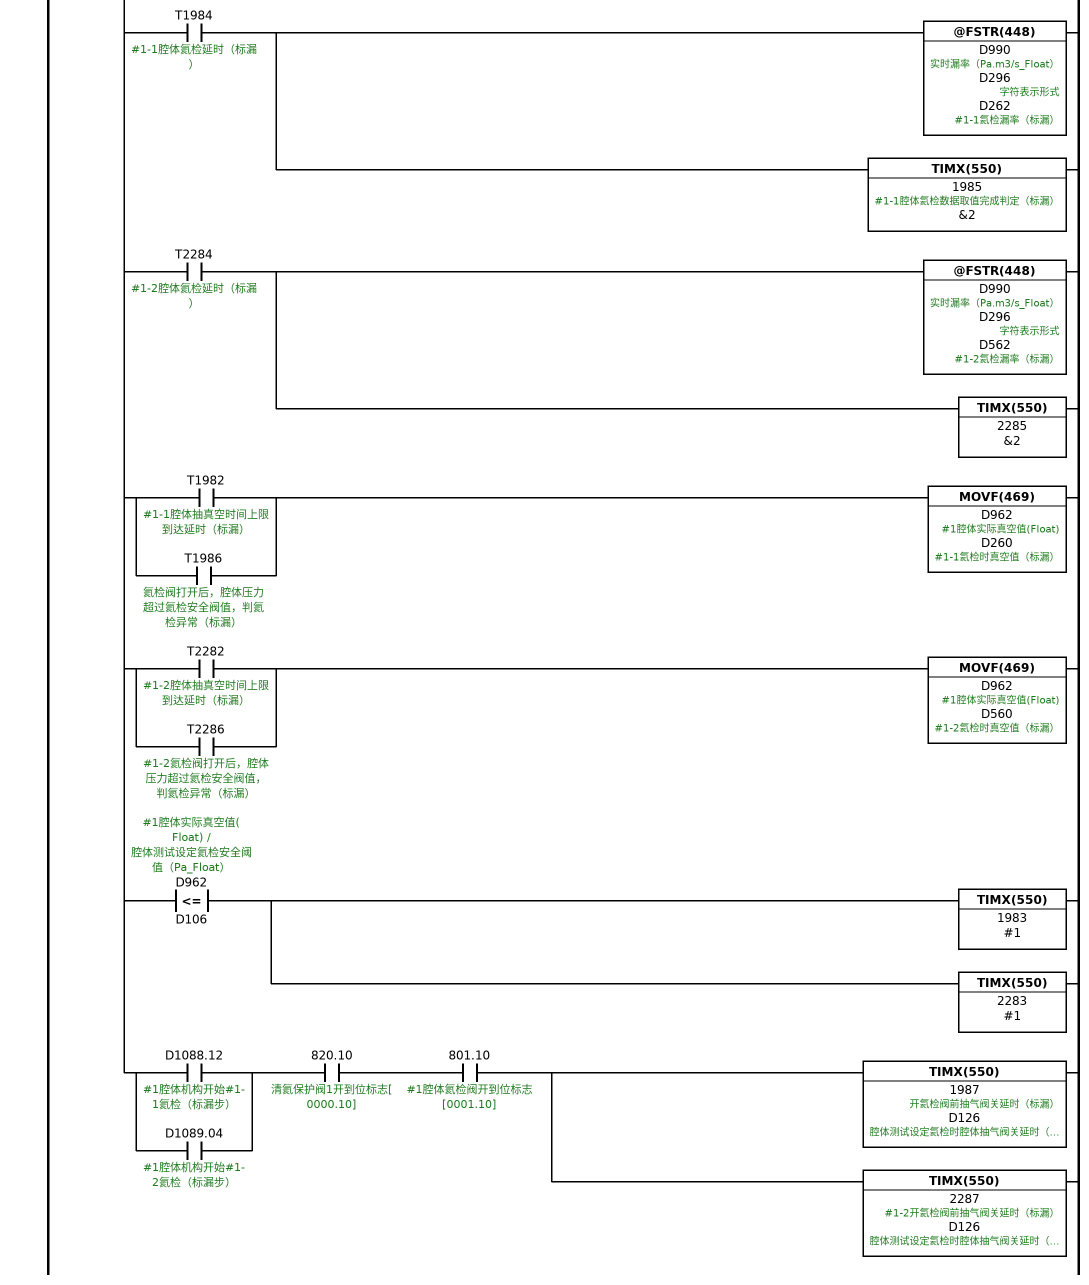
; rung 10: 标漏测试数据处理
LD P_On
OUT TR0
LD D1088.08  ; #1腔体机构开#1腔抽气阀（标漏步）
AND 821.00  ; #1腔体破真空挡板阀开到位标志
LD D1089.00  ; #1腔体机构开#1腔抽真空阀（标漏步）
AND 821.02  ; #1-2腔体阀开到位标志
ORLD
ANDLD
AND 820.14  ; #1腔体抽真空阀开到位标志
AND<=F(332) D962 D100  ; #1腔体实际真空值(Float), 腔体测试设定真空阈值（Pa_Float）
TIMX(550) 1981 &0  ; #1-1腔体抽真空阀值到达延时（标漏）
TIMX(550) 2281 &0  ; #1-2腔体抽真空阀值到达延时（标漏）
LD TR0
LD D1088.08  ; #1腔体机构开#1腔抽气阀（标漏步）
AND 821.00  ; #1腔体破真空挡板阀开到位标志
LD D1089.00  ; #1腔体机构开#1腔抽真空阀（标漏步）
AND 821.02  ; #1-2腔体阀开到位标志
ORLD
ANDLD
AND 820.14  ; #1腔体抽真空阀开到位标志
AND>F(333) D962 D100  ; #1腔体实际真空值(Float), 腔体测试设定真空阈值（Pa_Float）
TIMX(550) 1982 D102  ; 腔体测试设定抽真空时间上限（S_UInt）, #1-1腔体抽真空时间上限到达延时（标漏）
TIMX(550) 2282 D102  ; 腔体测试设定抽真空时间上限（S_UInt）, #1-2腔体抽真空时间上限到达延时（标漏）
LD TR0
AND D1088.12  ; #1腔体机构开始#1-1氦检（标漏步）
AND 821.00  ; #1腔体破真空挡板阀开到位标志
AND 820.10  ; 清氦保护阀1开到位标志[0000.10]
AND 801.10  ; #1腔体氦检阀开到位标志[0001.10]
TIMX(550) 1984 D110  ; 腔体测试设定氦检时间（S_UInt）, #1-1腔体氦检延时（标漏）
@MOVF(469) D962 D260  ; #1腔体实际真空值(Float), #1-1氦检时真空值（标漏）
AND>F(333) D962 D106  ; #1腔体实际真空值(Float), 腔体测试设定氦检安全阈值（Pa_Float）
TIMX(550) 1986 &0  ; 氦检阀打开后，腔体压力超过氦检安全阀值，判氦检异常（标漏）
LD TR0
AND D1089.04  ; #1腔体机构开始#1-2氦检（标漏步）
AND 821.02  ; #1-2腔体阀开到位标志
AND 820.10  ; 清氦保护阀1开到位标志[0000.10]
AND 801.10  ; #1腔体氦检阀开到位标志[0001.10]
TIMX(550) 2284 D110  ; 腔体测试设定氦检时间（S_UInt）, #1-2腔体氦检延时（标漏）
@MOVF(469) D962 D560  ; #1腔体实际真空值(Float), #1-2氦检时真空值（标漏）
AND>F(333) D962 D106  ; #1腔体实际真空值(Float), 腔体测试设定氦检安全阈值（Pa_Float）
TIMX(550) 2286 &0  ; #1-2氦检阀打开后，腔体压力超过氦检安全阀值，判氦检异常（标漏）
LD TR0
AND T1984  ; #1-1腔体氦检延时（标漏）
@FSTR(448) D990 D296 D262  ; 实时漏率（Pa.m3/s_Float）, 字符表示形式, #1-1氦检漏率（标漏）
TIMX(550) 1985 &2  ; #1-1腔体氦检数据取值完成判定（标漏）
LD TR0
AND T2284  ; #1-2腔体氦检延时（标漏）
@FSTR(448) D990 D296 D562  ; 实时漏率（Pa.m3/s_Float）, 字符表示形式, #1-2氦检漏率（标漏）
TIMX(550) 2285 &2
LD TR0
LD T1982  ; #1-1腔体抽真空时间上限到达延时（标漏）
OR T1986  ; 氦检阀打开后，腔体压力超过氦检安全阀值，判氦检异常（标漏）
ANDLD
MOVF(469) D962 D260  ; #1腔体实际真空值(Float), #1-1氦检时真空值（标漏）
LD TR0
LD T2282  ; #1-2腔体抽真空时间上限到达延时（标漏）
OR T2286  ; #1-2氦检阀打开后，腔体压力超过氦检安全阀值，判氦检异常（标漏）
ANDLD
MOVF(469) D962 D560  ; #1腔体实际真空值(Float), #1-2氦检时真空值（标漏）
LD TR0
AND<=F(332) D962 D106  ; #1腔体实际真空值(Float), 腔体测试设定氦检安全阈值（Pa_Float）
TIMX(550) 1983 #1
TIMX(550) 2283 #1
LD TR0
LD D1088.12  ; #1腔体机构开始#1-1氦检（标漏步）
OR D1089.04  ; #1腔体机构开始#1-2氦检（标漏步）
ANDLD
AND 820.10  ; 清氦保护阀1开到位标志[0000.10]
AND 801.10  ; #1腔体氦检阀开到位标志[0001.10]
TIMX(550) 1987 D126  ; 腔体测试设定氦检时腔体抽气阀关延时（S_UInt）, 开氦检阀前抽气阀关延时（标漏）
TIMX(550) 2287 D126  ; 腔体测试设定氦检时腔体抽气阀关延时（S_UInt）, #1-2开氦检阀前抽气阀关延时（标漏）
; rung 11: ********************** / #2腔体标漏流程 / **********************

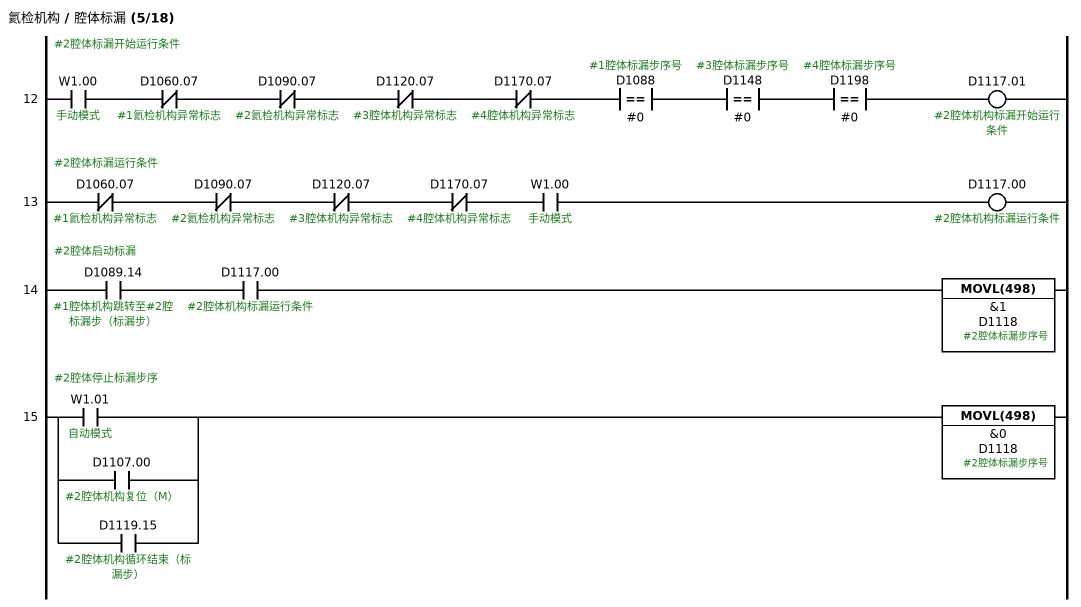
; rung 12: #2腔体标漏开始运行条件
LD W1.00  ; 手动模式
ANDNOT D1060.07  ; #1氦检机构异常标志
ANDNOT D1090.07  ; #2氦检机构异常标志
ANDNOT D1120.07  ; #3腔体机构异常标志
ANDNOT D1170.07  ; #4腔体机构异常标志
AND=L(301) D1088 #0  ; #1腔体标漏步序号
AND=L(301) D1148 #0  ; #3腔体标漏步序号
AND=L(301) D1198 #0  ; #4腔体标漏步序号
OUT D1117.01  ; #2腔体机构标漏开始运行条件
; rung 13: #2腔体标漏运行条件
LDNOT D1060.07  ; #1氦检机构异常标志
ANDNOT D1090.07  ; #2氦检机构异常标志
ANDNOT D1120.07  ; #3腔体机构异常标志
ANDNOT D1170.07  ; #4腔体机构异常标志
AND W1.00  ; 手动模式
OUT D1117.00  ; #2腔体机构标漏运行条件
; rung 14: #2腔体启动标漏
LD D1089.14  ; #1腔体机构跳转至#2腔标漏步（标漏步）
AND D1117.00  ; #2腔体机构标漏运行条件
MOVL(498) &1 D1118  ; #2腔体标漏步序号
; rung 15: #2腔体停止标漏步序
LD W1.01  ; 自动模式
OR D1107.00  ; #2腔体机构复位（M）
OR D1119.15  ; #2腔体机构循环结束（标漏步）
MOVL(498) &0 D1118  ; #2腔体标漏步序号

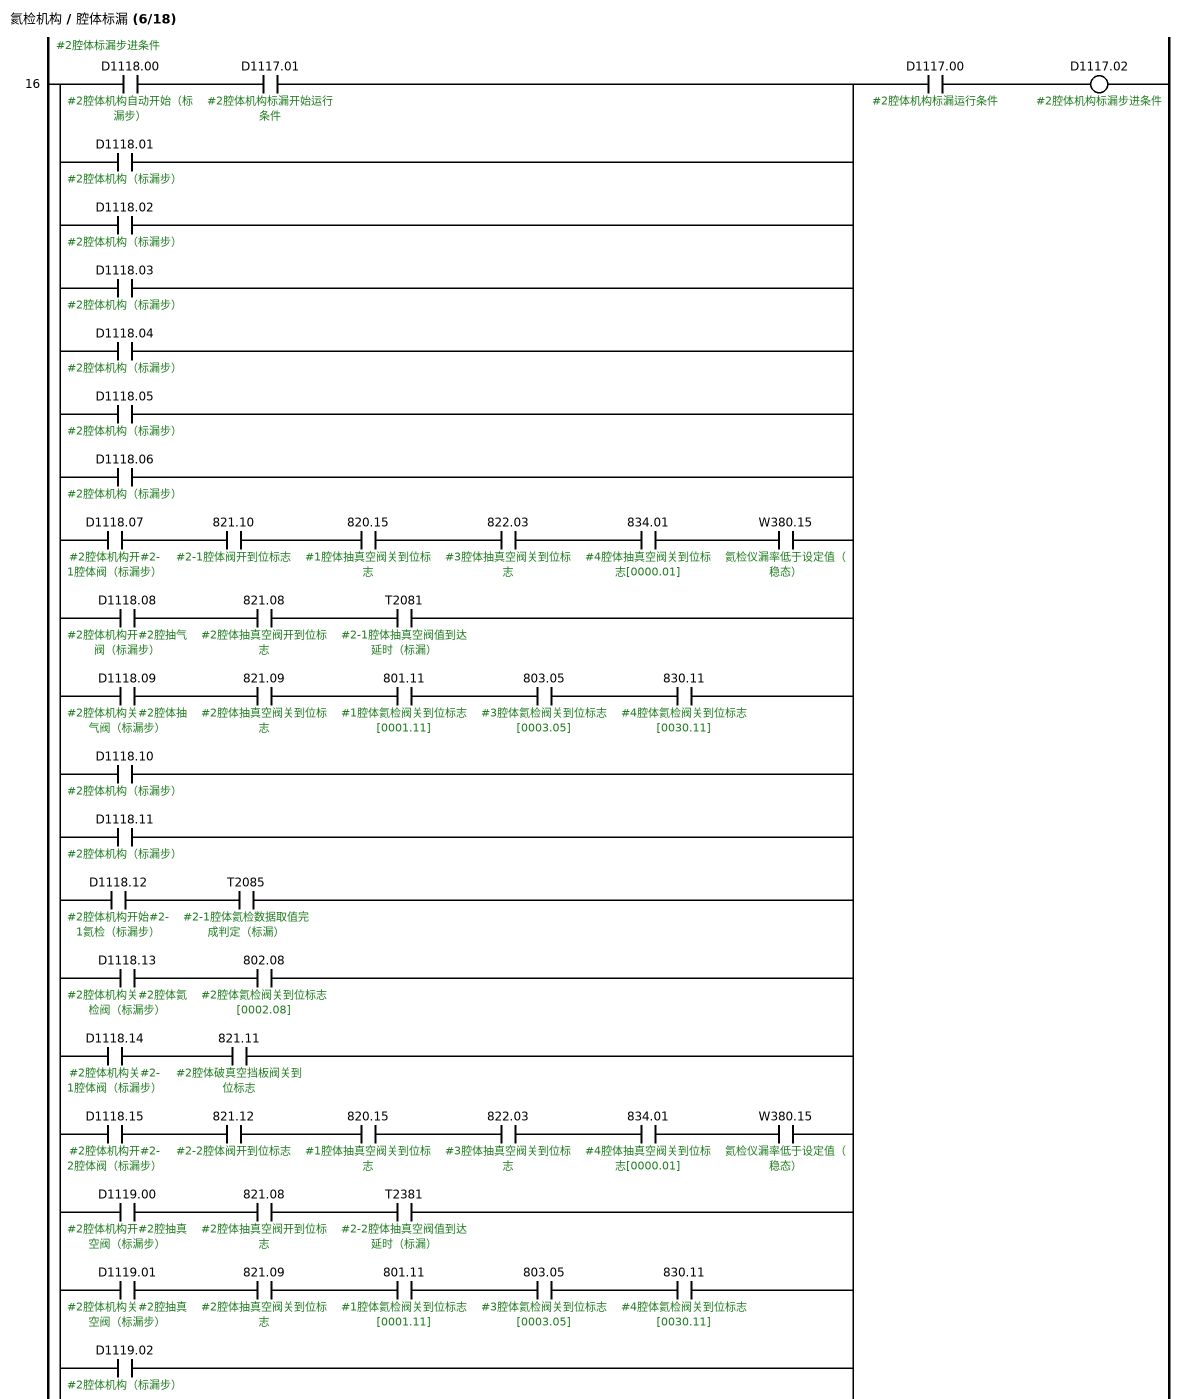

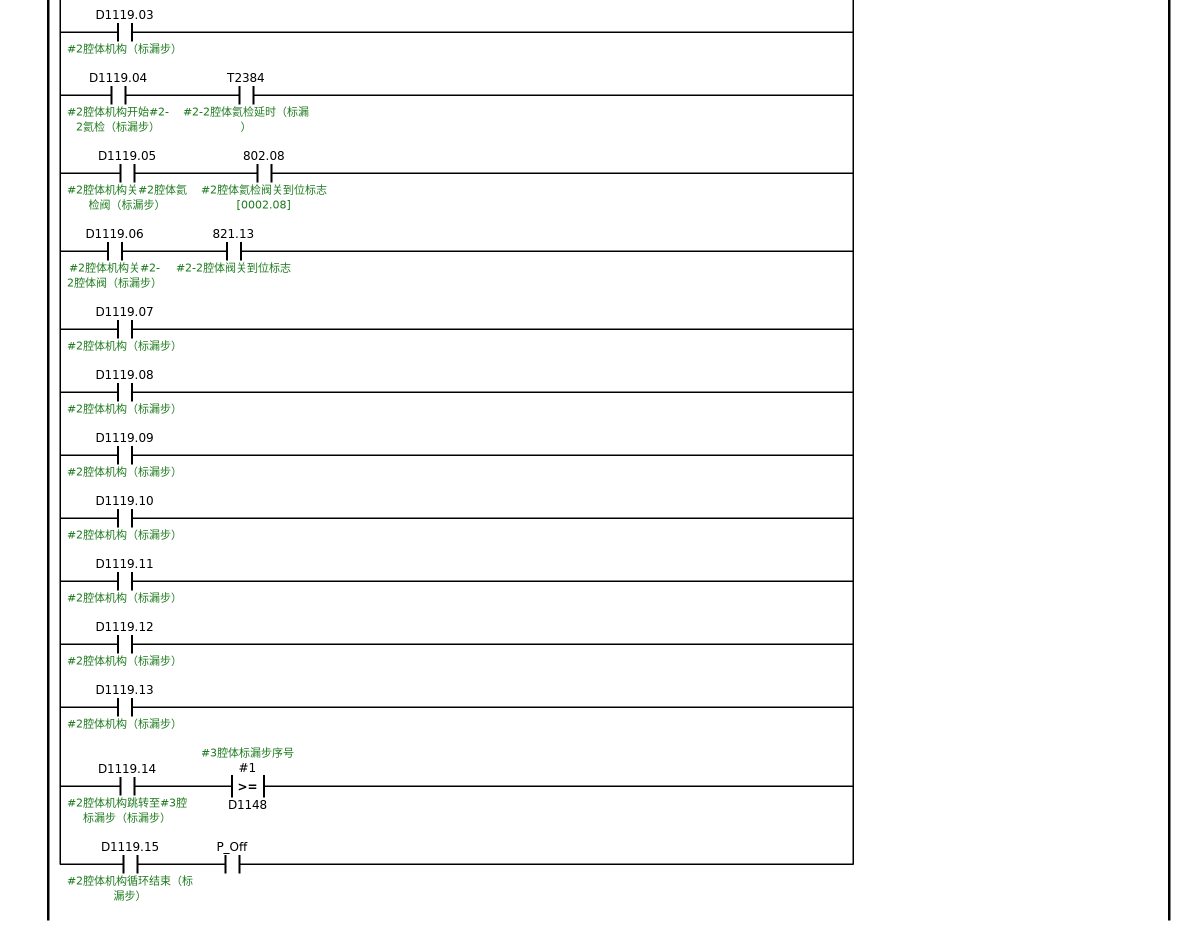
; rung 16: #2腔体标漏步进条件
LD D1118.00  ; #2腔体机构自动开始（标漏步）
AND D1117.01  ; #2腔体机构标漏开始运行条件
OR D1118.01  ; #2腔体机构（标漏步）
OR D1118.02  ; #2腔体机构（标漏步）
OR D1118.03  ; #2腔体机构（标漏步）
OR D1118.04  ; #2腔体机构（标漏步）
OR D1118.05  ; #2腔体机构（标漏步）
OR D1118.06  ; #2腔体机构（标漏步）
LD D1118.07  ; #2腔体机构开#2-1腔体阀（标漏步）
AND 821.10  ; #2-1腔体阀开到位标志
AND 820.15  ; #1腔体抽真空阀关到位标志
AND 822.03  ; #3腔体抽真空阀关到位标志
AND 834.01  ; #4腔体抽真空阀关到位标志[0000.01]
AND W380.15  ; 氦检仪漏率低于设定值（稳态）
ORLD
LD D1118.08  ; #2腔体机构开#2腔抽气阀（标漏步）
AND 821.08  ; #2腔体抽真空阀开到位标志
AND T2081  ; #2-1腔体抽真空阀值到达延时（标漏）
ORLD
LD D1118.09  ; #2腔体机构关#2腔体抽气阀（标漏步）
AND 821.09  ; #2腔体抽真空阀关到位标志
AND 801.11  ; #1腔体氦检阀关到位标志[0001.11]
AND 803.05  ; #3腔体氦检阀关到位标志[0003.05]
AND 830.11  ; #4腔体氦检阀关到位标志[0030.11]
ORLD
OR D1118.10  ; #2腔体机构（标漏步）
OR D1118.11  ; #2腔体机构（标漏步）
LD D1118.12  ; #2腔体机构开始#2-1氦检（标漏步）
AND T2085  ; #2-1腔体氦检数据取值完成判定（标漏）
ORLD
LD D1118.13  ; #2腔体机构关#2腔体氦检阀（标漏步）
AND 802.08  ; #2腔体氦检阀关到位标志[0002.08]
ORLD
LD D1118.14  ; #2腔体机构关#2-1腔体阀（标漏步）
AND 821.11  ; #2腔体破真空挡板阀关到位标志
ORLD
LD D1118.15  ; #2腔体机构开#2-2腔体阀（标漏步）
AND 821.12  ; #2-2腔体阀开到位标志
AND 820.15  ; #1腔体抽真空阀关到位标志
AND 822.03  ; #3腔体抽真空阀关到位标志
AND 834.01  ; #4腔体抽真空阀关到位标志[0000.01]
AND W380.15  ; 氦检仪漏率低于设定值（稳态）
ORLD
LD D1119.00  ; #2腔体机构开#2腔抽真空阀（标漏步）
AND 821.08  ; #2腔体抽真空阀开到位标志
AND T2381  ; #2-2腔体抽真空阀值到达延时（标漏）
ORLD
LD D1119.01  ; #2腔体机构关#2腔抽真空阀（标漏步）
AND 821.09  ; #2腔体抽真空阀关到位标志
AND 801.11  ; #1腔体氦检阀关到位标志[0001.11]
AND 803.05  ; #3腔体氦检阀关到位标志[0003.05]
AND 830.11  ; #4腔体氦检阀关到位标志[0030.11]
ORLD
OR D1119.02  ; #2腔体机构（标漏步）
OR D1119.03  ; #2腔体机构（标漏步）
LD D1119.04  ; #2腔体机构开始#2-2氦检（标漏步）
AND T2384  ; #2-2腔体氦检延时（标漏）
ORLD
LD D1119.05  ; #2腔体机构关#2腔体氦检阀（标漏步）
AND 802.08  ; #2腔体氦检阀关到位标志[0002.08]
ORLD
LD D1119.06  ; #2腔体机构关#2-2腔体阀（标漏步）
AND 821.13  ; #2-2腔体阀关到位标志
ORLD
OR D1119.07  ; #2腔体机构（标漏步）
OR D1119.08  ; #2腔体机构（标漏步）
OR D1119.09  ; #2腔体机构（标漏步）
OR D1119.10  ; #2腔体机构（标漏步）
OR D1119.11  ; #2腔体机构（标漏步）
OR D1119.12  ; #2腔体机构（标漏步）
OR D1119.13  ; #2腔体机构（标漏步）
LD D1119.14  ; #2腔体机构跳转至#3腔标漏步（标漏步）
AND>=L(326) #1 D1148  ; #3腔体标漏步序号
ORLD
LD D1119.15  ; #2腔体机构循环结束（标漏步）
AND P_Off
ORLD
AND D1117.00  ; #2腔体机构标漏运行条件
OUT D1117.02  ; #2腔体机构标漏步进条件

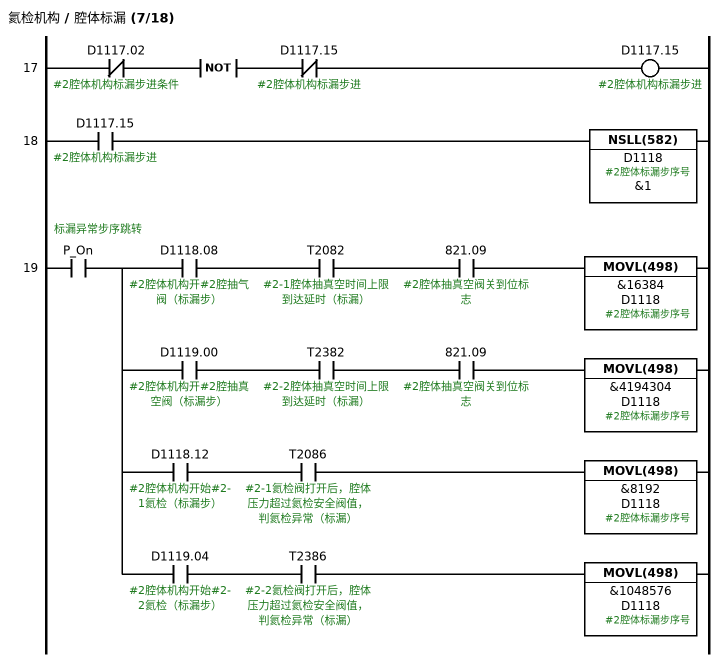
; rung 17
LDNOT D1117.02  ; #2腔体机构标漏步进条件
NOT(520)
ANDNOT D1117.15  ; #2腔体机构标漏步进
OUT D1117.15  ; #2腔体机构标漏步进
; rung 18
LD D1117.15  ; #2腔体机构标漏步进
NSLL(582) D1118 &1  ; #2腔体标漏步序号
; rung 19: 标漏异常步序跳转
LD P_On
OUT TR0
AND D1118.08  ; #2腔体机构开#2腔抽气阀（标漏步）
AND T2082  ; #2-1腔体抽真空时间上限到达延时（标漏）
AND 821.09  ; #2腔体抽真空阀关到位标志
MOVL(498) &16384 D1118  ; #2腔体标漏步序号
LD TR0
AND D1119.00  ; #2腔体机构开#2腔抽真空阀（标漏步）
AND T2382  ; #2-2腔体抽真空时间上限到达延时（标漏）
AND 821.09  ; #2腔体抽真空阀关到位标志
MOVL(498) &4194304 D1118  ; #2腔体标漏步序号
LD TR0
AND D1118.12  ; #2腔体机构开始#2-1氦检（标漏步）
AND T2086  ; #2-1氦检阀打开后，腔体压力超过氦检安全阀值，判氦检异常（标漏）
MOVL(498) &8192 D1118  ; #2腔体标漏步序号
LD TR0
AND D1119.04  ; #2腔体机构开始#2-2氦检（标漏步）
AND T2386  ; #2-2氦检阀打开后，腔体压力超过氦检安全阀值，判氦检异常（标漏）
MOVL(498) &1048576 D1118  ; #2腔体标漏步序号

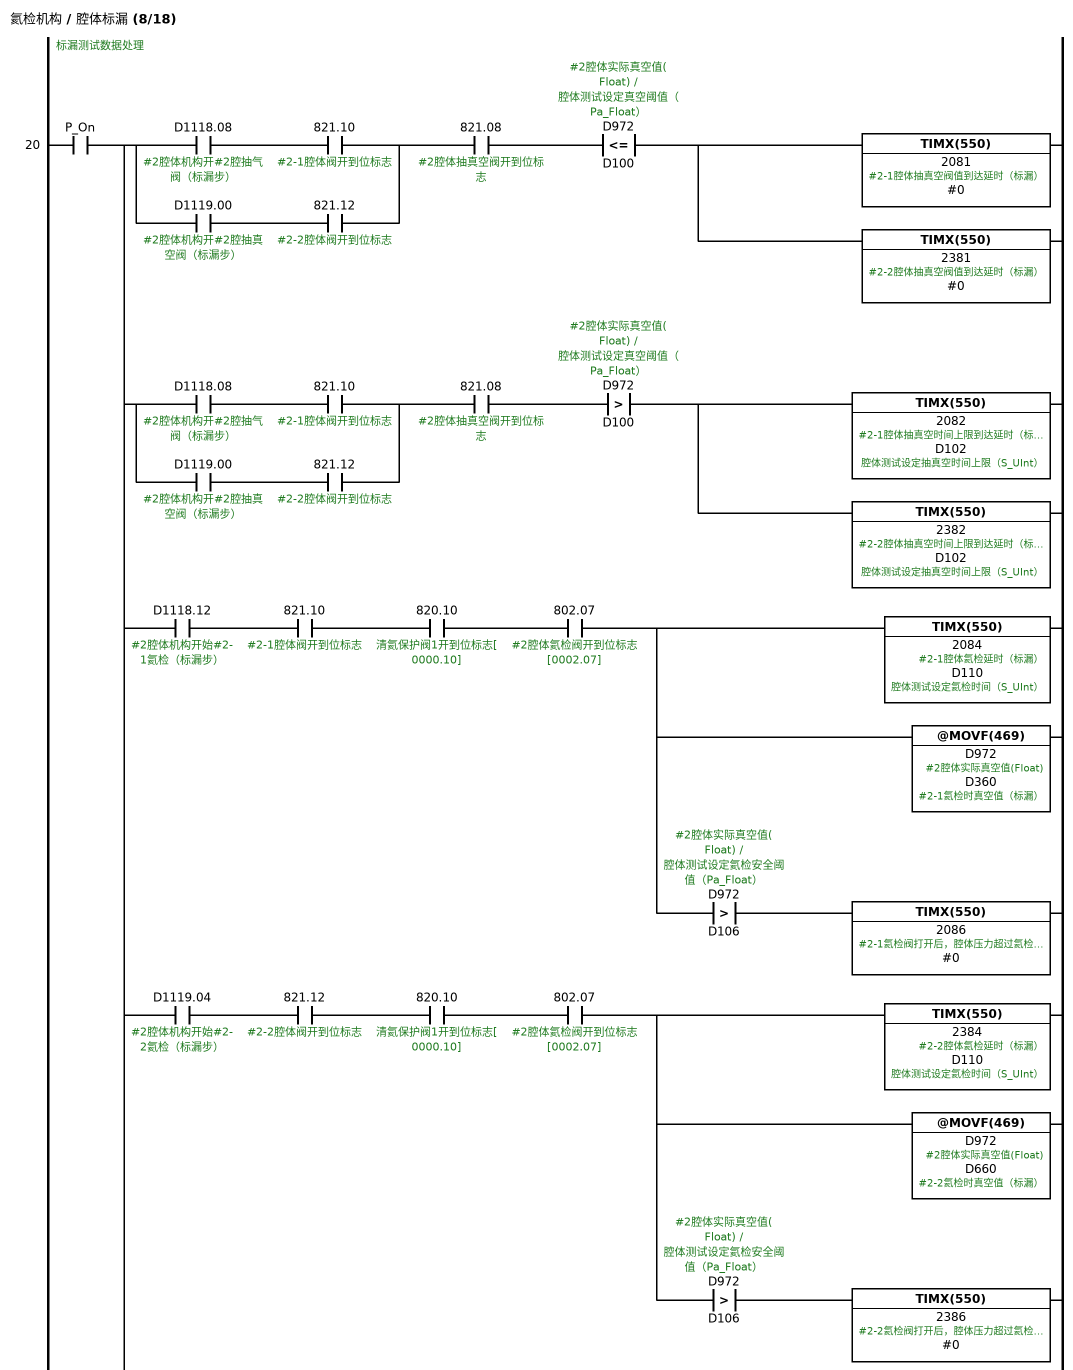

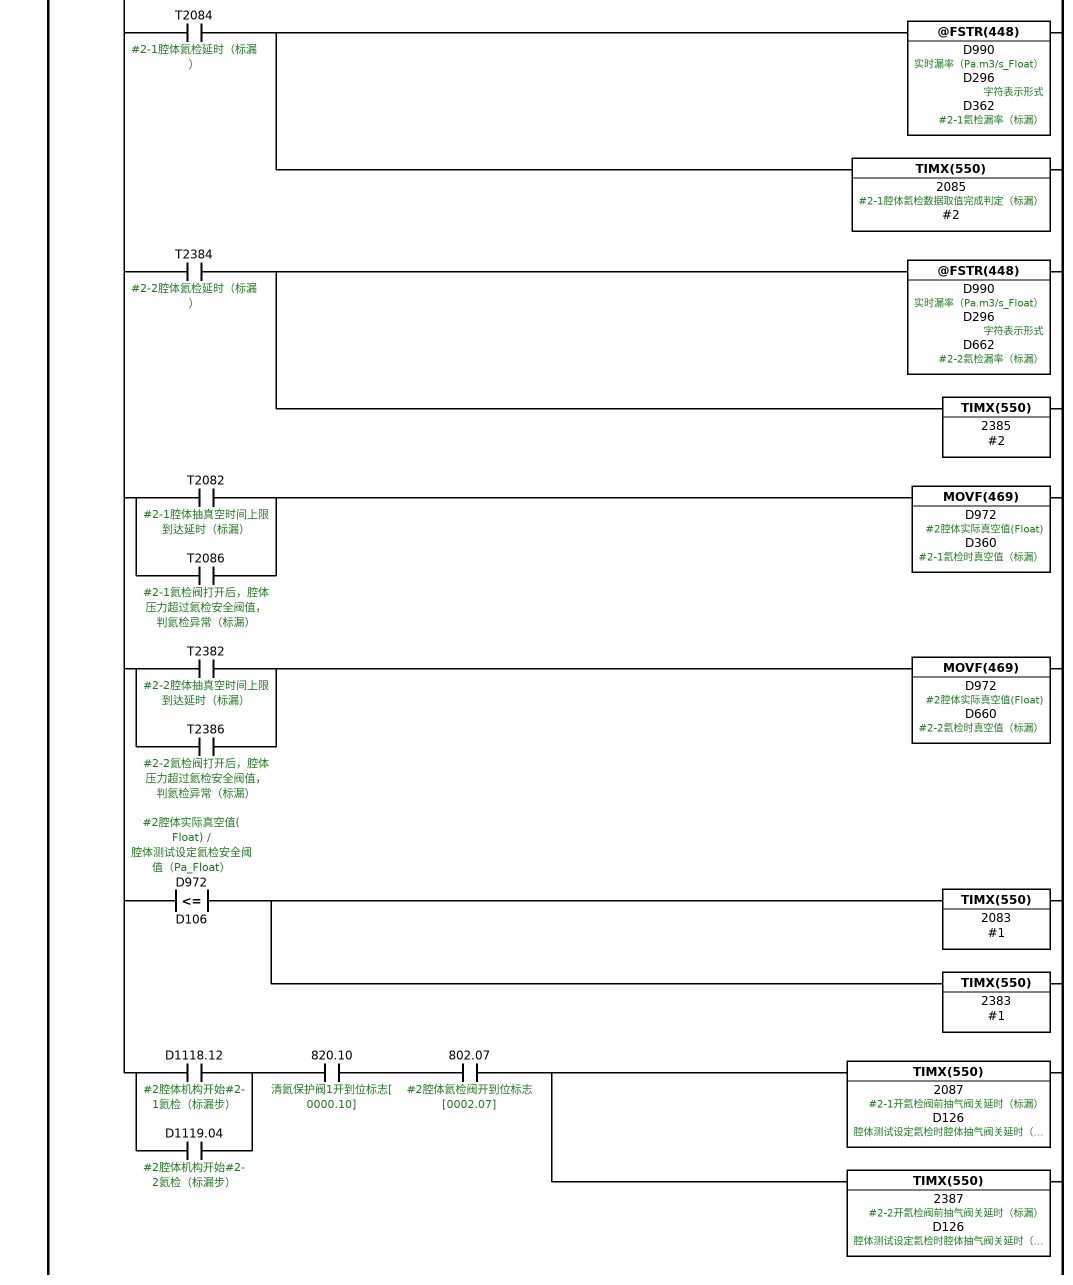
; rung 20: 标漏测试数据处理
LD P_On
OUT TR0
LD D1118.08  ; #2腔体机构开#2腔抽气阀（标漏步）
AND 821.10  ; #2-1腔体阀开到位标志
LD D1119.00  ; #2腔体机构开#2腔抽真空阀（标漏步）
AND 821.12  ; #2-2腔体阀开到位标志
ORLD
ANDLD
AND 821.08  ; #2腔体抽真空阀开到位标志
AND<=F(332) D972 D100  ; #2腔体实际真空值(Float), 腔体测试设定真空阈值（Pa_Float）
TIMX(550) 2081 #0  ; #2-1腔体抽真空阀值到达延时（标漏）
TIMX(550) 2381 #0  ; #2-2腔体抽真空阀值到达延时（标漏）
LD TR0
LD D1118.08  ; #2腔体机构开#2腔抽气阀（标漏步）
AND 821.10  ; #2-1腔体阀开到位标志
LD D1119.00  ; #2腔体机构开#2腔抽真空阀（标漏步）
AND 821.12  ; #2-2腔体阀开到位标志
ORLD
ANDLD
AND 821.08  ; #2腔体抽真空阀开到位标志
AND>F(333) D972 D100  ; #2腔体实际真空值(Float), 腔体测试设定真空阈值（Pa_Float）
TIMX(550) 2082 D102  ; 腔体测试设定抽真空时间上限（S_UInt）, #2-1腔体抽真空时间上限到达延时（标漏）
TIMX(550) 2382 D102  ; 腔体测试设定抽真空时间上限（S_UInt）, #2-2腔体抽真空时间上限到达延时（标漏）
LD TR0
AND D1118.12  ; #2腔体机构开始#2-1氦检（标漏步）
AND 821.10  ; #2-1腔体阀开到位标志
AND 820.10  ; 清氦保护阀1开到位标志[0000.10]
AND 802.07  ; #2腔体氦检阀开到位标志[0002.07]
TIMX(550) 2084 D110  ; 腔体测试设定氦检时间（S_UInt）, #2-1腔体氦检延时（标漏）
@MOVF(469) D972 D360  ; #2腔体实际真空值(Float), #2-1氦检时真空值（标漏）
AND>F(333) D972 D106  ; #2腔体实际真空值(Float), 腔体测试设定氦检安全阈值（Pa_Float）
TIMX(550) 2086 #0  ; #2-1氦检阀打开后，腔体压力超过氦检安全阀值，判氦检异常（标漏）
LD TR0
AND D1119.04  ; #2腔体机构开始#2-2氦检（标漏步）
AND 821.12  ; #2-2腔体阀开到位标志
AND 820.10  ; 清氦保护阀1开到位标志[0000.10]
AND 802.07  ; #2腔体氦检阀开到位标志[0002.07]
TIMX(550) 2384 D110  ; 腔体测试设定氦检时间（S_UInt）, #2-2腔体氦检延时（标漏）
@MOVF(469) D972 D660  ; #2腔体实际真空值(Float), #2-2氦检时真空值（标漏）
AND>F(333) D972 D106  ; #2腔体实际真空值(Float), 腔体测试设定氦检安全阈值（Pa_Float）
TIMX(550) 2386 #0  ; #2-2氦检阀打开后，腔体压力超过氦检安全阀值，判氦检异常（标漏）
LD TR0
AND T2084  ; #2-1腔体氦检延时（标漏）
@FSTR(448) D990 D296 D362  ; 实时漏率（Pa.m3/s_Float）, 字符表示形式, #2-1氦检漏率（标漏）
TIMX(550) 2085 #2  ; #2-1腔体氦检数据取值完成判定（标漏）
LD TR0
AND T2384  ; #2-2腔体氦检延时（标漏）
@FSTR(448) D990 D296 D662  ; 实时漏率（Pa.m3/s_Float）, 字符表示形式, #2-2氦检漏率（标漏）
TIMX(550) 2385 #2
LD TR0
LD T2082  ; #2-1腔体抽真空时间上限到达延时（标漏）
OR T2086  ; #2-1氦检阀打开后，腔体压力超过氦检安全阀值，判氦检异常（标漏）
ANDLD
MOVF(469) D972 D360  ; #2腔体实际真空值(Float), #2-1氦检时真空值（标漏）
LD TR0
LD T2382  ; #2-2腔体抽真空时间上限到达延时（标漏）
OR T2386  ; #2-2氦检阀打开后，腔体压力超过氦检安全阀值，判氦检异常（标漏）
ANDLD
MOVF(469) D972 D660  ; #2腔体实际真空值(Float), #2-2氦检时真空值（标漏）
LD TR0
AND<=F(332) D972 D106  ; #2腔体实际真空值(Float), 腔体测试设定氦检安全阈值（Pa_Float）
TIMX(550) 2083 #1
TIMX(550) 2383 #1
LD TR0
LD D1118.12  ; #2腔体机构开始#2-1氦检（标漏步）
OR D1119.04  ; #2腔体机构开始#2-2氦检（标漏步）
ANDLD
AND 820.10  ; 清氦保护阀1开到位标志[0000.10]
AND 802.07  ; #2腔体氦检阀开到位标志[0002.07]
TIMX(550) 2087 D126  ; 腔体测试设定氦检时腔体抽气阀关延时（S_UInt）, #2-1开氦检阀前抽气阀关延时（标漏）
TIMX(550) 2387 D126  ; 腔体测试设定氦检时腔体抽气阀关延时（S_UInt）, #2-2开氦检阀前抽气阀关延时（标漏）
; rung 21: ********************** / #3腔体标漏流程 / **********************

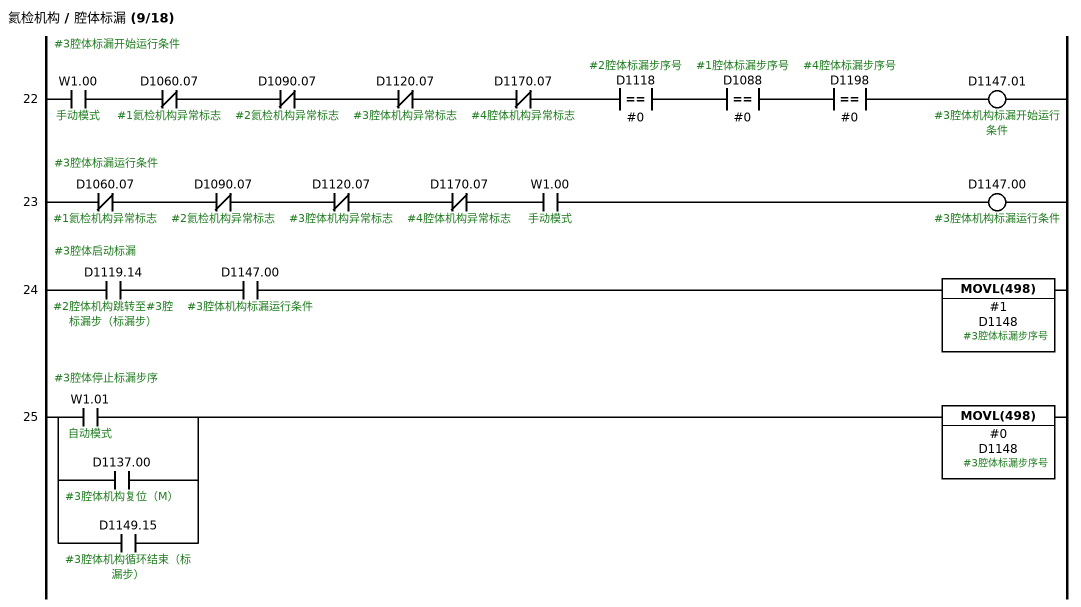
; rung 22: #3腔体标漏开始运行条件
LD W1.00  ; 手动模式
ANDNOT D1060.07  ; #1氦检机构异常标志
ANDNOT D1090.07  ; #2氦检机构异常标志
ANDNOT D1120.07  ; #3腔体机构异常标志
ANDNOT D1170.07  ; #4腔体机构异常标志
AND=L(301) D1118 #0  ; #2腔体标漏步序号
AND=L(301) D1088 #0  ; #1腔体标漏步序号
AND=L(301) D1198 #0  ; #4腔体标漏步序号
OUT D1147.01  ; #3腔体机构标漏开始运行条件
; rung 23: #3腔体标漏运行条件
LDNOT D1060.07  ; #1氦检机构异常标志
ANDNOT D1090.07  ; #2氦检机构异常标志
ANDNOT D1120.07  ; #3腔体机构异常标志
ANDNOT D1170.07  ; #4腔体机构异常标志
AND W1.00  ; 手动模式
OUT D1147.00  ; #3腔体机构标漏运行条件
; rung 24: #3腔体启动标漏
LD D1119.14  ; #2腔体机构跳转至#3腔标漏步（标漏步）
AND D1147.00  ; #3腔体机构标漏运行条件
MOVL(498) #1 D1148  ; #3腔体标漏步序号
; rung 25: #3腔体停止标漏步序
LD W1.01  ; 自动模式
OR D1137.00  ; #3腔体机构复位（M）
OR D1149.15  ; #3腔体机构循环结束（标漏步）
MOVL(498) #0 D1148  ; #3腔体标漏步序号

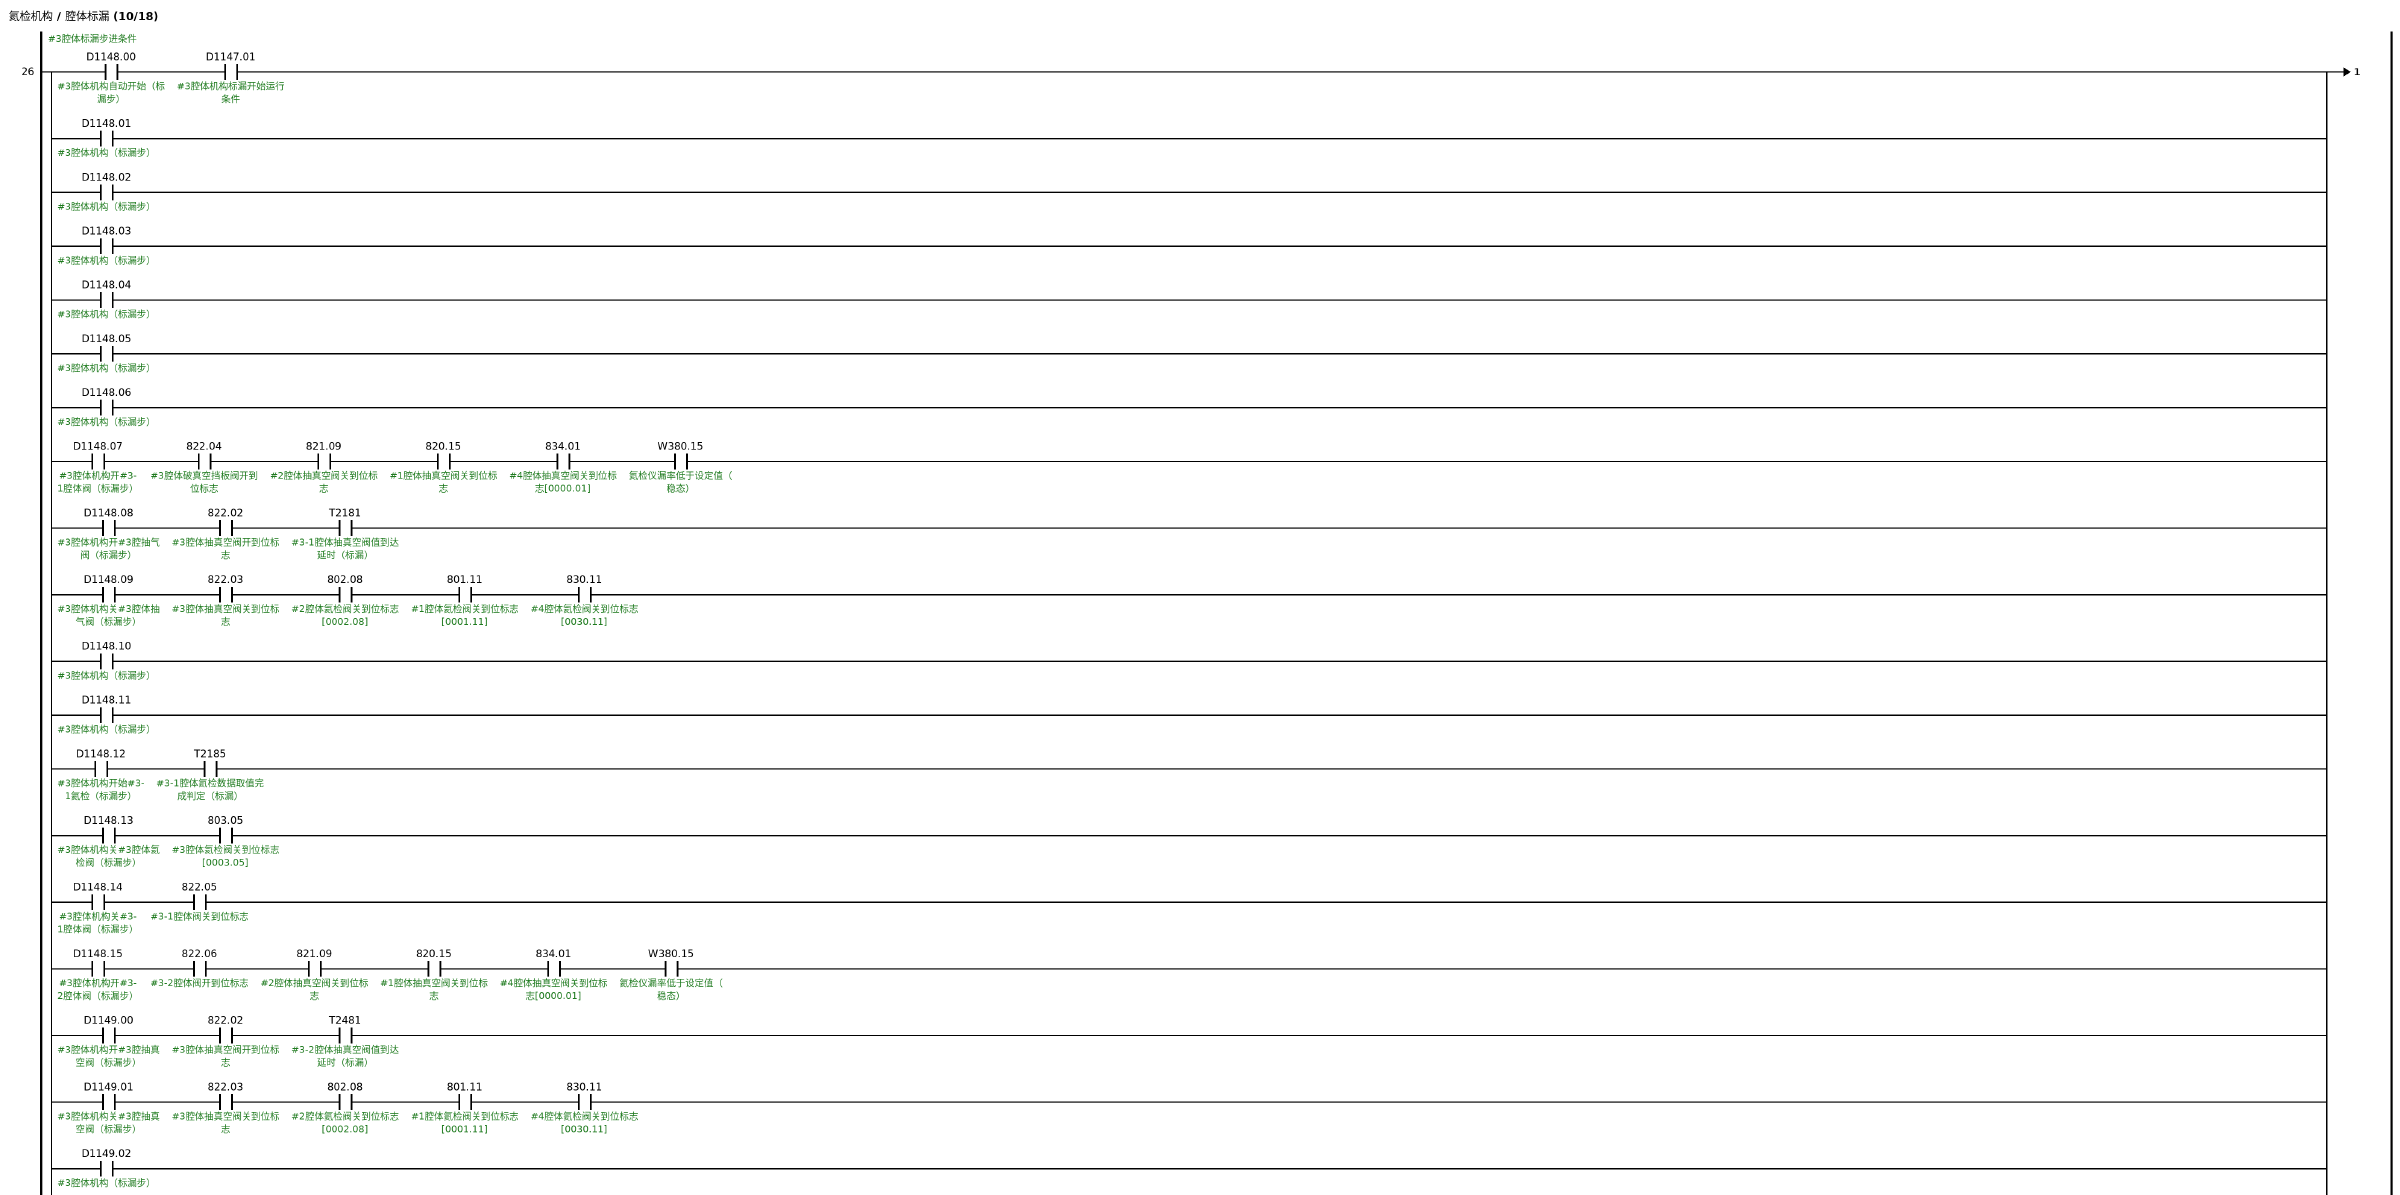

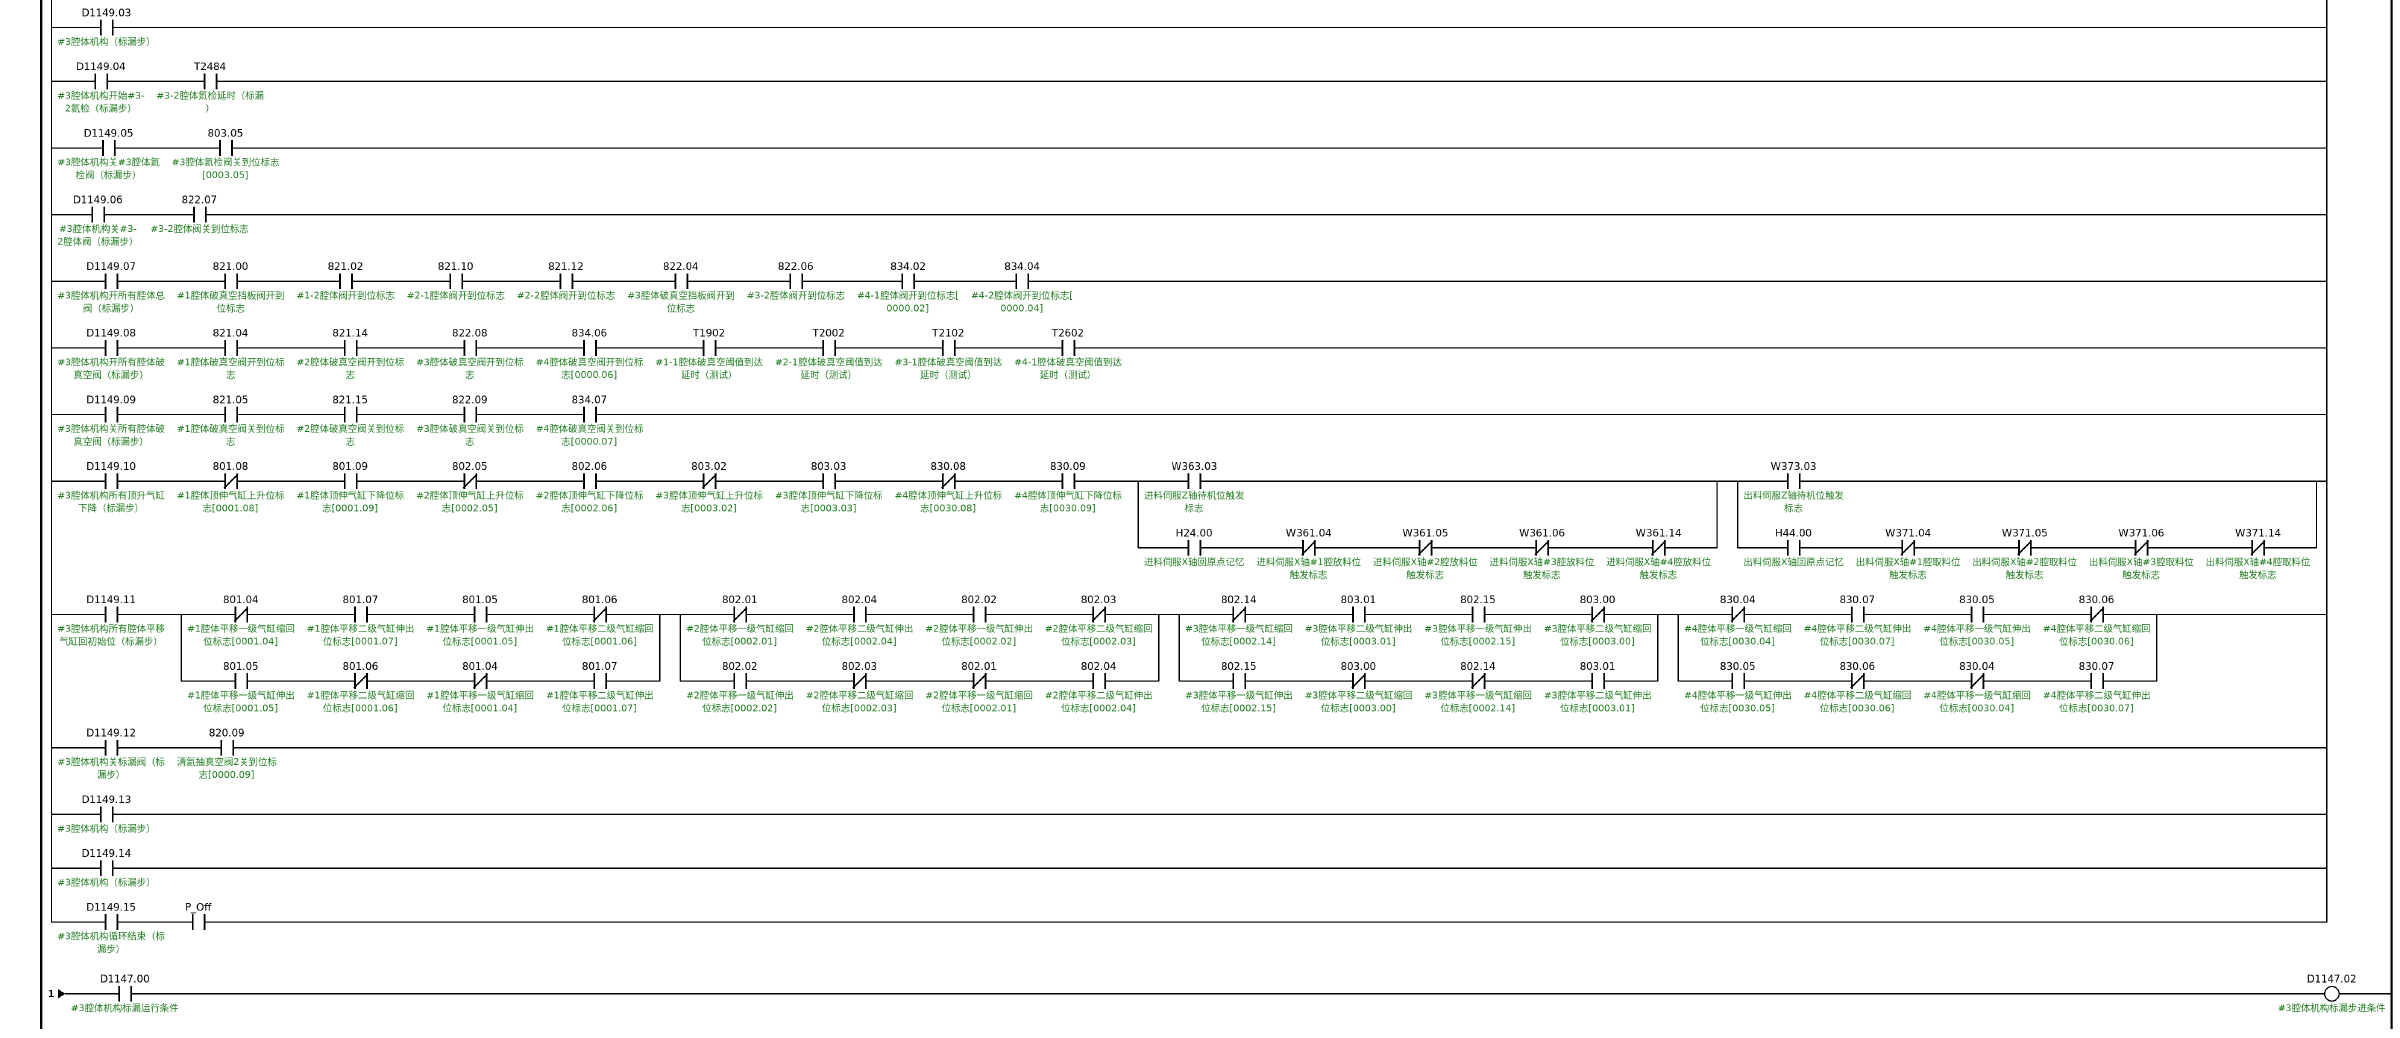
; rung 26: #3腔体标漏步进条件
LD D1148.00  ; #3腔体机构自动开始（标漏步）
AND D1147.01  ; #3腔体机构标漏开始运行条件
OR D1148.01  ; #3腔体机构（标漏步）
OR D1148.02  ; #3腔体机构（标漏步）
OR D1148.03  ; #3腔体机构（标漏步）
OR D1148.04  ; #3腔体机构（标漏步）
OR D1148.05  ; #3腔体机构（标漏步）
OR D1148.06  ; #3腔体机构（标漏步）
LD D1148.07  ; #3腔体机构开#3-1腔体阀（标漏步）
AND 822.04  ; #3腔体破真空挡板阀开到位标志
AND 821.09  ; #2腔体抽真空阀关到位标志
AND 820.15  ; #1腔体抽真空阀关到位标志
AND 834.01  ; #4腔体抽真空阀关到位标志[0000.01]
AND W380.15  ; 氦检仪漏率低于设定值（稳态）
ORLD
LD D1148.08  ; #3腔体机构开#3腔抽气阀（标漏步）
AND 822.02  ; #3腔体抽真空阀开到位标志
AND T2181  ; #3-1腔体抽真空阀值到达延时（标漏）
ORLD
LD D1148.09  ; #3腔体机构关#3腔体抽气阀（标漏步）
AND 822.03  ; #3腔体抽真空阀关到位标志
AND 802.08  ; #2腔体氦检阀关到位标志[0002.08]
AND 801.11  ; #1腔体氦检阀关到位标志[0001.11]
AND 830.11  ; #4腔体氦检阀关到位标志[0030.11]
ORLD
OR D1148.10  ; #3腔体机构（标漏步）
OR D1148.11  ; #3腔体机构（标漏步）
LD D1148.12  ; #3腔体机构开始#3-1氦检（标漏步）
AND T2185  ; #3-1腔体氦检数据取值完成判定（标漏）
ORLD
LD D1148.13  ; #3腔体机构关#3腔体氦检阀（标漏步）
AND 803.05  ; #3腔体氦检阀关到位标志[0003.05]
ORLD
LD D1148.14  ; #3腔体机构关#3-1腔体阀（标漏步）
AND 822.05  ; #3-1腔体阀关到位标志
ORLD
LD D1148.15  ; #3腔体机构开#3-2腔体阀（标漏步）
AND 822.06  ; #3-2腔体阀开到位标志
AND 821.09  ; #2腔体抽真空阀关到位标志
AND 820.15  ; #1腔体抽真空阀关到位标志
AND 834.01  ; #4腔体抽真空阀关到位标志[0000.01]
AND W380.15  ; 氦检仪漏率低于设定值（稳态）
ORLD
LD D1149.00  ; #3腔体机构开#3腔抽真空阀（标漏步）
AND 822.02  ; #3腔体抽真空阀开到位标志
AND T2481  ; #3-2腔体抽真空阀值到达延时（标漏）
ORLD
LD D1149.01  ; #3腔体机构关#3腔抽真空阀（标漏步）
AND 822.03  ; #3腔体抽真空阀关到位标志
AND 802.08  ; #2腔体氦检阀关到位标志[0002.08]
AND 801.11  ; #1腔体氦检阀关到位标志[0001.11]
AND 830.11  ; #4腔体氦检阀关到位标志[0030.11]
ORLD
OR D1149.02  ; #3腔体机构（标漏步）
OR D1149.03  ; #3腔体机构（标漏步）
LD D1149.04  ; #3腔体机构开始#3-2氦检（标漏步）
AND T2484  ; #3-2腔体氦检延时（标漏）
ORLD
LD D1149.05  ; #3腔体机构关#3腔体氦检阀（标漏步）
AND 803.05  ; #3腔体氦检阀关到位标志[0003.05]
ORLD
LD D1149.06  ; #3腔体机构关#3-2腔体阀（标漏步）
AND 822.07  ; #3-2腔体阀关到位标志
ORLD
LD D1149.07  ; #3腔体机构开所有腔体总阀（标漏步）
AND 821.00  ; #1腔体破真空挡板阀开到位标志
AND 821.02  ; #1-2腔体阀开到位标志
AND 821.10  ; #2-1腔体阀开到位标志
AND 821.12  ; #2-2腔体阀开到位标志
AND 822.04  ; #3腔体破真空挡板阀开到位标志
AND 822.06  ; #3-2腔体阀开到位标志
AND 834.02  ; #4-1腔体阀开到位标志[0000.02]
AND 834.04  ; #4-2腔体阀开到位标志[0000.04]
ORLD
LD D1149.08  ; #3腔体机构开所有腔体破真空阀（标漏步）
AND 821.04  ; #1腔体破真空阀开到位标志
AND 821.14  ; #2腔体破真空阀开到位标志
AND 822.08  ; #3腔体破真空阀开到位标志
AND 834.06  ; #4腔体破真空阀开到位标志[0000.06]
AND T1902  ; #1-1腔体破真空阈值到达延时（测试）
AND T2002  ; #2-1腔体破真空阈值到达延时（测试）
AND T2102  ; #3-1腔体破真空阈值到达延时（测试）
AND T2602  ; #4-1腔体破真空阈值到达延时（测试）
ORLD
LD D1149.09  ; #3腔体机构关所有腔体破真空阀（标漏步）
AND 821.05  ; #1腔体破真空阀关到位标志
AND 821.15  ; #2腔体破真空阀关到位标志
AND 822.09  ; #3腔体破真空阀关到位标志
AND 834.07  ; #4腔体破真空阀关到位标志[0000.07]
ORLD
LD D1149.10  ; #3腔体机构所有顶升气缸下降（标漏步）
ANDNOT 801.08  ; #1腔体顶伸气缸上升位标志[0001.08]
AND 801.09  ; #1腔体顶伸气缸下降位标志[0001.09]
ANDNOT 802.05  ; #2腔体顶伸气缸上升位标志[0002.05]
AND 802.06  ; #2腔体顶伸气缸下降位标志[0002.06]
ANDNOT 803.02  ; #3腔体顶伸气缸上升位标志[0003.02]
AND 803.03  ; #3腔体顶伸气缸下降位标志[0003.03]
ANDNOT 830.08  ; #4腔体顶伸气缸上升位标志[0030.08]
AND 830.09  ; #4腔体顶伸气缸下降位标志[0030.09]
LD W363.03  ; 进料伺服Z轴待机位触发标志
LD H24.00  ; 进料伺服X轴回原点记忆
ANDNOT W361.04  ; 进料伺服X轴#1腔放料位触发标志
ANDNOT W361.05  ; 进料伺服X轴#2腔放料位触发标志
ANDNOT W361.06  ; 进料伺服X轴#3腔放料位触发标志
ANDNOT W361.14  ; 进料伺服X轴#4腔放料位触发标志
ORLD
ANDLD
LD W373.03  ; 出料伺服Z轴待机位触发标志
LD H44.00  ; 出料伺服X轴回原点记忆
ANDNOT W371.04  ; 出料伺服X轴#1腔取料位触发标志
ANDNOT W371.05  ; 出料伺服X轴#2腔取料位触发标志
ANDNOT W371.06  ; 出料伺服X轴#3腔取料位触发标志
ANDNOT W371.14  ; 出料伺服X轴#4腔取料位触发标志
ORLD
ANDLD
ORLD
LD D1149.11  ; #3腔体机构所有腔体平移气缸回初始位（标漏步）
LDNOT 801.04  ; #1腔体平移一级气缸缩回位标志[0001.04]
AND 801.07  ; #1腔体平移二级气缸伸出位标志[0001.07]
AND 801.05  ; #1腔体平移一级气缸伸出位标志[0001.05]
ANDNOT 801.06  ; #1腔体平移二级气缸缩回位标志[0001.06]
LD 801.05  ; #1腔体平移一级气缸伸出位标志[0001.05]
ANDNOT 801.06  ; #1腔体平移二级气缸缩回位标志[0001.06]
ANDNOT 801.04  ; #1腔体平移一级气缸缩回位标志[0001.04]
AND 801.07  ; #1腔体平移二级气缸伸出位标志[0001.07]
ORLD
ANDLD
LDNOT 802.01  ; #2腔体平移一级气缸缩回位标志[0002.01]
AND 802.04  ; #2腔体平移二级气缸伸出位标志[0002.04]
AND 802.02  ; #2腔体平移一级气缸伸出位标志[0002.02]
ANDNOT 802.03  ; #2腔体平移二级气缸缩回位标志[0002.03]
LD 802.02  ; #2腔体平移一级气缸伸出位标志[0002.02]
ANDNOT 802.03  ; #2腔体平移二级气缸缩回位标志[0002.03]
ANDNOT 802.01  ; #2腔体平移一级气缸缩回位标志[0002.01]
AND 802.04  ; #2腔体平移二级气缸伸出位标志[0002.04]
ORLD
ANDLD
LDNOT 802.14  ; #3腔体平移一级气缸缩回位标志[0002.14]
AND 803.01  ; #3腔体平移二级气缸伸出位标志[0003.01]
AND 802.15  ; #3腔体平移一级气缸伸出位标志[0002.15]
ANDNOT 803.00  ; #3腔体平移二级气缸缩回位标志[0003.00]
LD 802.15  ; #3腔体平移一级气缸伸出位标志[0002.15]
ANDNOT 803.00  ; #3腔体平移二级气缸缩回位标志[0003.00]
ANDNOT 802.14  ; #3腔体平移一级气缸缩回位标志[0002.14]
AND 803.01  ; #3腔体平移二级气缸伸出位标志[0003.01]
ORLD
ANDLD
LDNOT 830.04  ; #4腔体平移一级气缸缩回位标志[0030.04]
AND 830.07  ; #4腔体平移二级气缸伸出位标志[0030.07]
AND 830.05  ; #4腔体平移一级气缸伸出位标志[0030.05]
ANDNOT 830.06  ; #4腔体平移二级气缸缩回位标志[0030.06]
LD 830.05  ; #4腔体平移一级气缸伸出位标志[0030.05]
ANDNOT 830.06  ; #4腔体平移二级气缸缩回位标志[0030.06]
ANDNOT 830.04  ; #4腔体平移一级气缸缩回位标志[0030.04]
AND 830.07  ; #4腔体平移二级气缸伸出位标志[0030.07]
ORLD
ANDLD
ORLD
LD D1149.12  ; #3腔体机构关标漏阀（标漏步）
AND 820.09  ; 清氦抽真空阀2关到位标志[0000.09]
ORLD
OR D1149.13  ; #3腔体机构（标漏步）
OR D1149.14  ; #3腔体机构（标漏步）
LD D1149.15  ; #3腔体机构循环结束（标漏步）
AND P_Off
ORLD
AND D1147.00  ; #3腔体机构标漏运行条件
OUT D1147.02  ; #3腔体机构标漏步进条件

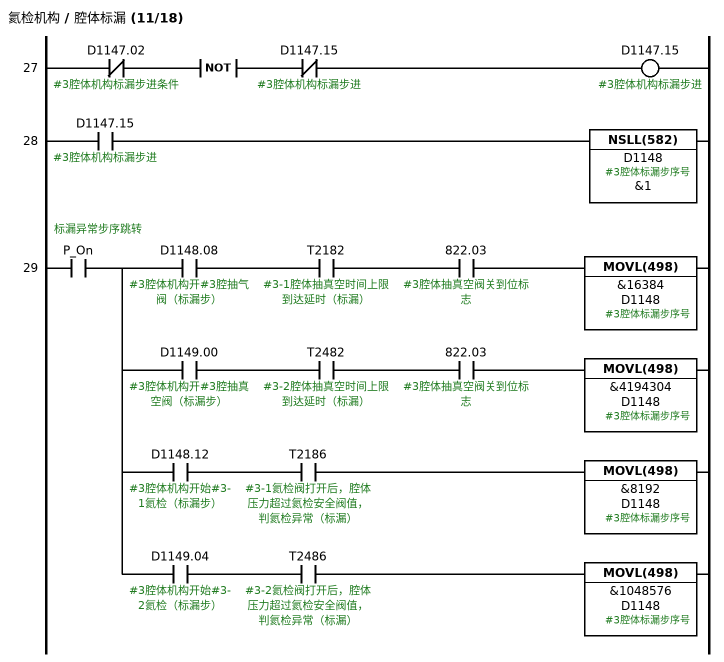
; rung 27
LDNOT D1147.02  ; #3腔体机构标漏步进条件
NOT(520)
ANDNOT D1147.15  ; #3腔体机构标漏步进
OUT D1147.15  ; #3腔体机构标漏步进
; rung 28
LD D1147.15  ; #3腔体机构标漏步进
NSLL(582) D1148 &1  ; #3腔体标漏步序号
; rung 29: 标漏异常步序跳转
LD P_On
OUT TR0
AND D1148.08  ; #3腔体机构开#3腔抽气阀（标漏步）
AND T2182  ; #3-1腔体抽真空时间上限到达延时（标漏）
AND 822.03  ; #3腔体抽真空阀关到位标志
MOVL(498) &16384 D1148  ; #3腔体标漏步序号
LD TR0
AND D1149.00  ; #3腔体机构开#3腔抽真空阀（标漏步）
AND T2482  ; #3-2腔体抽真空时间上限到达延时（标漏）
AND 822.03  ; #3腔体抽真空阀关到位标志
MOVL(498) &4194304 D1148  ; #3腔体标漏步序号
LD TR0
AND D1148.12  ; #3腔体机构开始#3-1氦检（标漏步）
AND T2186  ; #3-1氦检阀打开后，腔体压力超过氦检安全阀值，判氦检异常（标漏）
MOVL(498) &8192 D1148  ; #3腔体标漏步序号
LD TR0
AND D1149.04  ; #3腔体机构开始#3-2氦检（标漏步）
AND T2486  ; #3-2氦检阀打开后，腔体压力超过氦检安全阀值，判氦检异常（标漏）
MOVL(498) &1048576 D1148  ; #3腔体标漏步序号

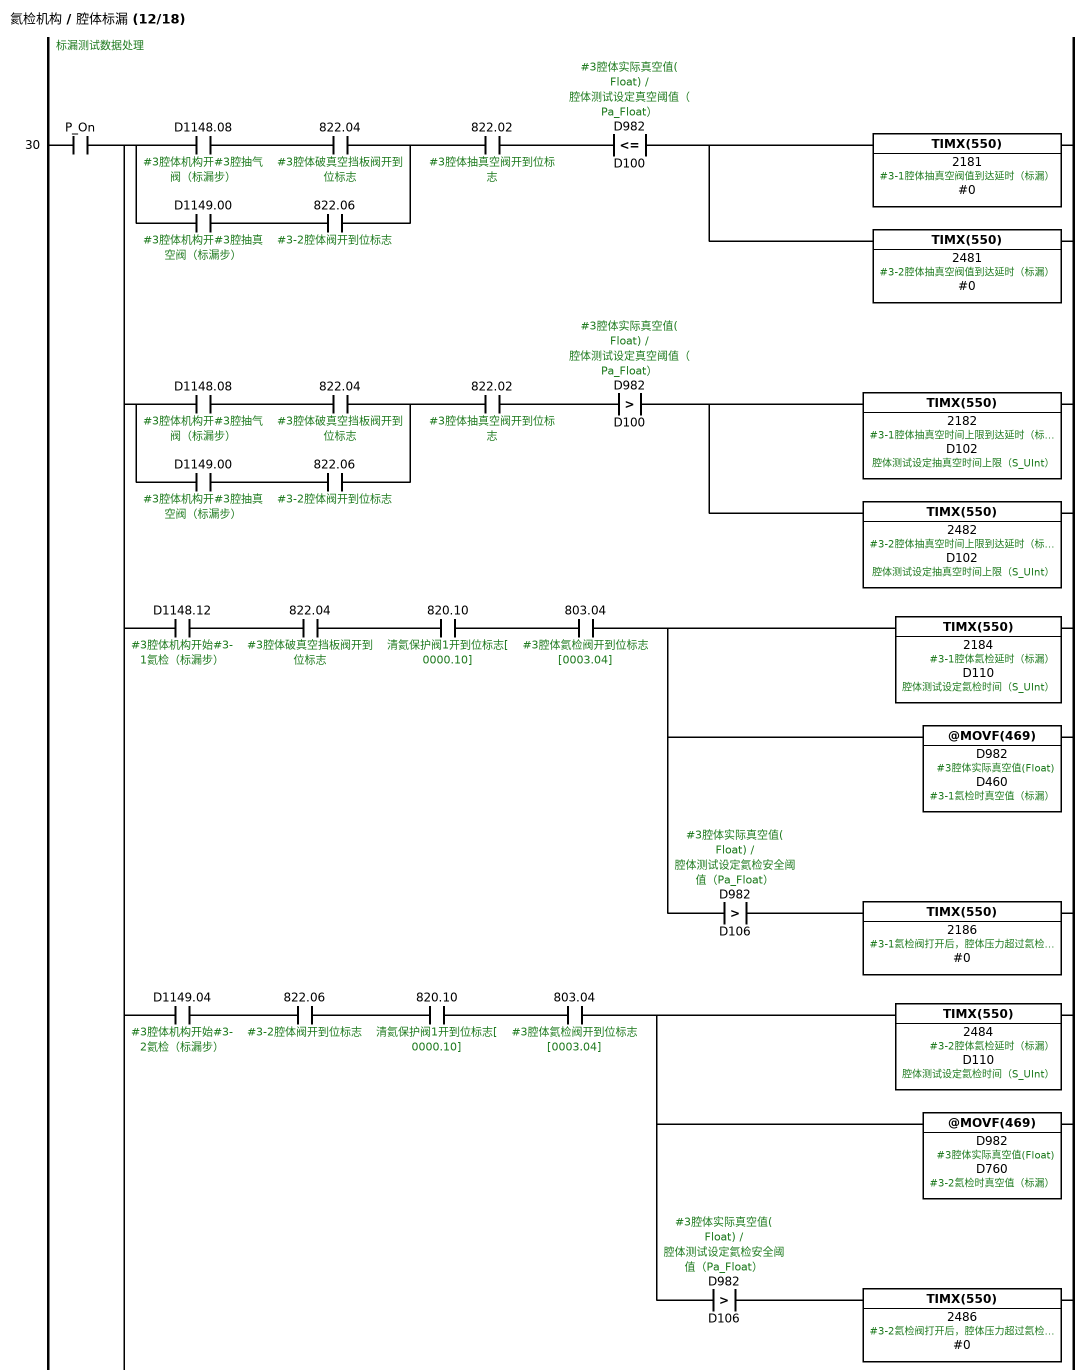

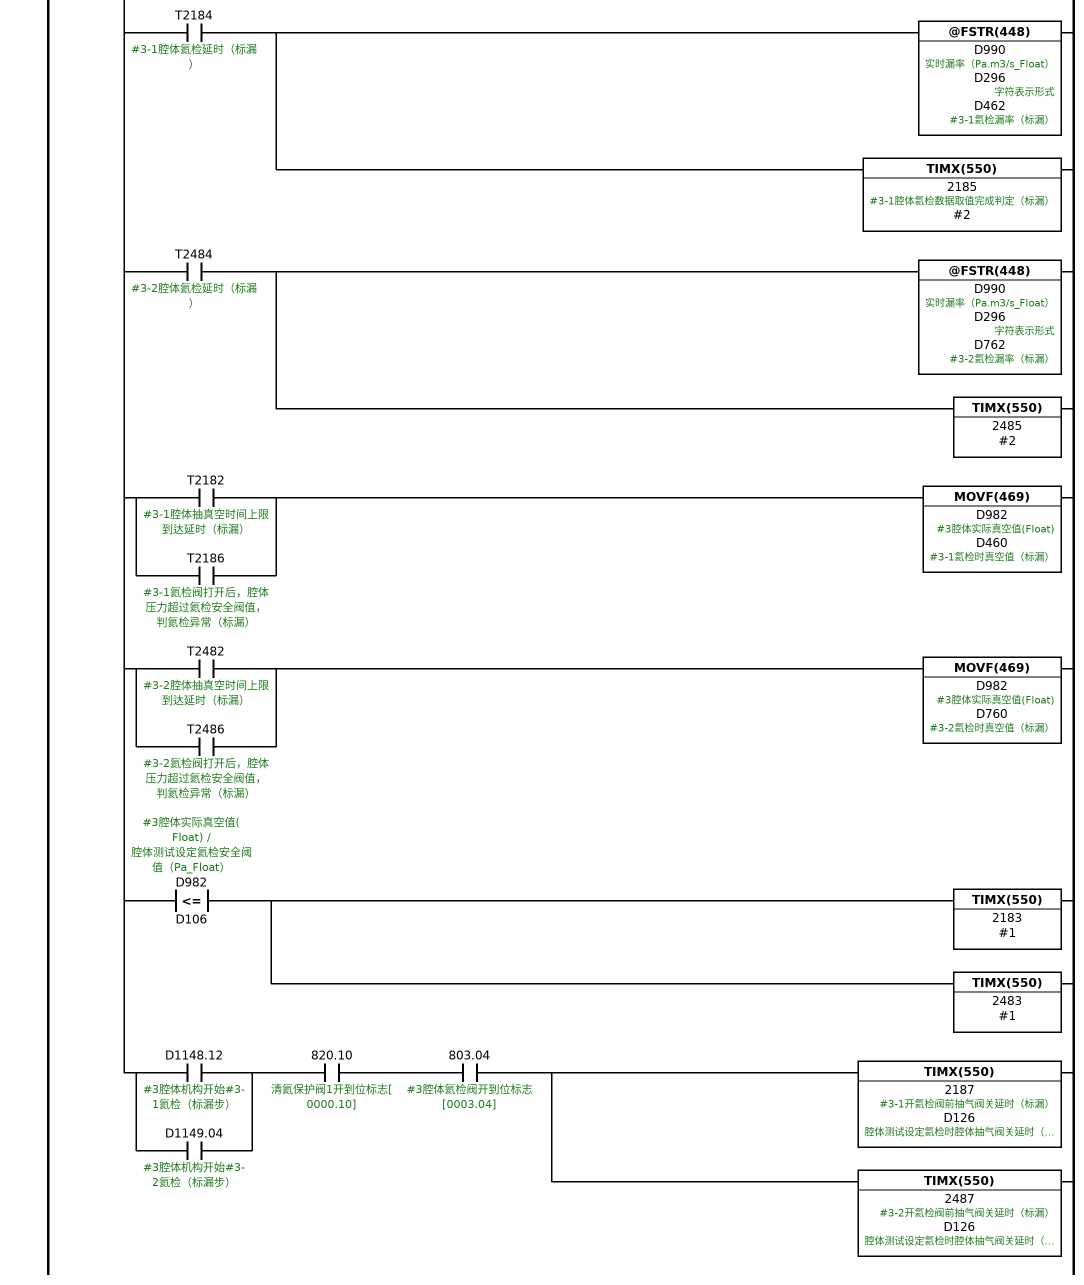
; rung 30: 标漏测试数据处理
LD P_On
OUT TR0
LD D1148.08  ; #3腔体机构开#3腔抽气阀（标漏步）
AND 822.04  ; #3腔体破真空挡板阀开到位标志
LD D1149.00  ; #3腔体机构开#3腔抽真空阀（标漏步）
AND 822.06  ; #3-2腔体阀开到位标志
ORLD
ANDLD
AND 822.02  ; #3腔体抽真空阀开到位标志
AND<=F(332) D982 D100  ; #3腔体实际真空值(Float), 腔体测试设定真空阈值（Pa_Float）
TIMX(550) 2181 #0  ; #3-1腔体抽真空阀值到达延时（标漏）
TIMX(550) 2481 #0  ; #3-2腔体抽真空阀值到达延时（标漏）
LD TR0
LD D1148.08  ; #3腔体机构开#3腔抽气阀（标漏步）
AND 822.04  ; #3腔体破真空挡板阀开到位标志
LD D1149.00  ; #3腔体机构开#3腔抽真空阀（标漏步）
AND 822.06  ; #3-2腔体阀开到位标志
ORLD
ANDLD
AND 822.02  ; #3腔体抽真空阀开到位标志
AND>F(333) D982 D100  ; #3腔体实际真空值(Float), 腔体测试设定真空阈值（Pa_Float）
TIMX(550) 2182 D102  ; 腔体测试设定抽真空时间上限（S_UInt）, #3-1腔体抽真空时间上限到达延时（标漏）
TIMX(550) 2482 D102  ; 腔体测试设定抽真空时间上限（S_UInt）, #3-2腔体抽真空时间上限到达延时（标漏）
LD TR0
AND D1148.12  ; #3腔体机构开始#3-1氦检（标漏步）
AND 822.04  ; #3腔体破真空挡板阀开到位标志
AND 820.10  ; 清氦保护阀1开到位标志[0000.10]
AND 803.04  ; #3腔体氦检阀开到位标志[0003.04]
TIMX(550) 2184 D110  ; 腔体测试设定氦检时间（S_UInt）, #3-1腔体氦检延时（标漏）
@MOVF(469) D982 D460  ; #3腔体实际真空值(Float), #3-1氦检时真空值（标漏）
AND>F(333) D982 D106  ; #3腔体实际真空值(Float), 腔体测试设定氦检安全阈值（Pa_Float）
TIMX(550) 2186 #0  ; #3-1氦检阀打开后，腔体压力超过氦检安全阀值，判氦检异常（标漏）
LD TR0
AND D1149.04  ; #3腔体机构开始#3-2氦检（标漏步）
AND 822.06  ; #3-2腔体阀开到位标志
AND 820.10  ; 清氦保护阀1开到位标志[0000.10]
AND 803.04  ; #3腔体氦检阀开到位标志[0003.04]
TIMX(550) 2484 D110  ; 腔体测试设定氦检时间（S_UInt）, #3-2腔体氦检延时（标漏）
@MOVF(469) D982 D760  ; #3腔体实际真空值(Float), #3-2氦检时真空值（标漏）
AND>F(333) D982 D106  ; #3腔体实际真空值(Float), 腔体测试设定氦检安全阈值（Pa_Float）
TIMX(550) 2486 #0  ; #3-2氦检阀打开后，腔体压力超过氦检安全阀值，判氦检异常（标漏）
LD TR0
AND T2184  ; #3-1腔体氦检延时（标漏）
@FSTR(448) D990 D296 D462  ; 实时漏率（Pa.m3/s_Float）, 字符表示形式, #3-1氦检漏率（标漏）
TIMX(550) 2185 #2  ; #3-1腔体氦检数据取值完成判定（标漏）
LD TR0
AND T2484  ; #3-2腔体氦检延时（标漏）
@FSTR(448) D990 D296 D762  ; 实时漏率（Pa.m3/s_Float）, 字符表示形式, #3-2氦检漏率（标漏）
TIMX(550) 2485 #2
LD TR0
LD T2182  ; #3-1腔体抽真空时间上限到达延时（标漏）
OR T2186  ; #3-1氦检阀打开后，腔体压力超过氦检安全阀值，判氦检异常（标漏）
ANDLD
MOVF(469) D982 D460  ; #3腔体实际真空值(Float), #3-1氦检时真空值（标漏）
LD TR0
LD T2482  ; #3-2腔体抽真空时间上限到达延时（标漏）
OR T2486  ; #3-2氦检阀打开后，腔体压力超过氦检安全阀值，判氦检异常（标漏）
ANDLD
MOVF(469) D982 D760  ; #3腔体实际真空值(Float), #3-2氦检时真空值（标漏）
LD TR0
AND<=F(332) D982 D106  ; #3腔体实际真空值(Float), 腔体测试设定氦检安全阈值（Pa_Float）
TIMX(550) 2183 #1
TIMX(550) 2483 #1
LD TR0
LD D1148.12  ; #3腔体机构开始#3-1氦检（标漏步）
OR D1149.04  ; #3腔体机构开始#3-2氦检（标漏步）
ANDLD
AND 820.10  ; 清氦保护阀1开到位标志[0000.10]
AND 803.04  ; #3腔体氦检阀开到位标志[0003.04]
TIMX(550) 2187 D126  ; 腔体测试设定氦检时腔体抽气阀关延时（S_UInt）, #3-1开氦检阀前抽气阀关延时（标漏）
TIMX(550) 2487 D126  ; 腔体测试设定氦检时腔体抽气阀关延时（S_UInt）, #3-2开氦检阀前抽气阀关延时（标漏）
; rung 31: ********************** / #4腔体标漏流程 / **********************

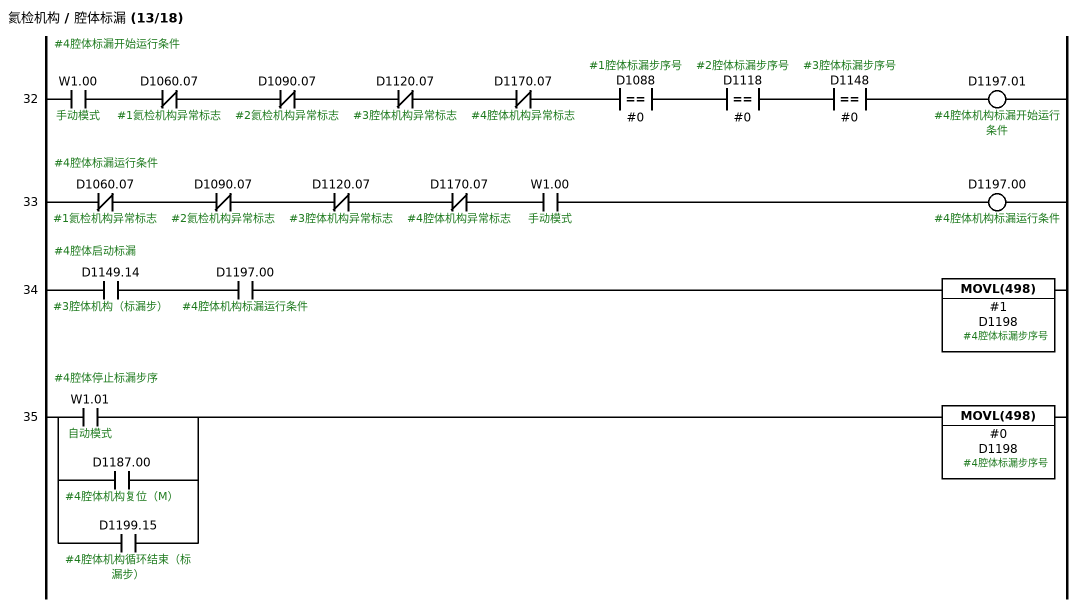
; rung 32: #4腔体标漏开始运行条件
LD W1.00  ; 手动模式
ANDNOT D1060.07  ; #1氦检机构异常标志
ANDNOT D1090.07  ; #2氦检机构异常标志
ANDNOT D1120.07  ; #3腔体机构异常标志
ANDNOT D1170.07  ; #4腔体机构异常标志
AND=L(301) D1088 #0  ; #1腔体标漏步序号
AND=L(301) D1118 #0  ; #2腔体标漏步序号
AND=L(301) D1148 #0  ; #3腔体标漏步序号
OUT D1197.01  ; #4腔体机构标漏开始运行条件
; rung 33: #4腔体标漏运行条件
LDNOT D1060.07  ; #1氦检机构异常标志
ANDNOT D1090.07  ; #2氦检机构异常标志
ANDNOT D1120.07  ; #3腔体机构异常标志
ANDNOT D1170.07  ; #4腔体机构异常标志
AND W1.00  ; 手动模式
OUT D1197.00  ; #4腔体机构标漏运行条件
; rung 34: #4腔体启动标漏
LD D1149.14  ; #3腔体机构（标漏步）
AND D1197.00  ; #4腔体机构标漏运行条件
MOVL(498) #1 D1198  ; #4腔体标漏步序号
; rung 35: #4腔体停止标漏步序
LD W1.01  ; 自动模式
OR D1187.00  ; #4腔体机构复位（M）
OR D1199.15  ; #4腔体机构循环结束（标漏步）
MOVL(498) #0 D1198  ; #4腔体标漏步序号

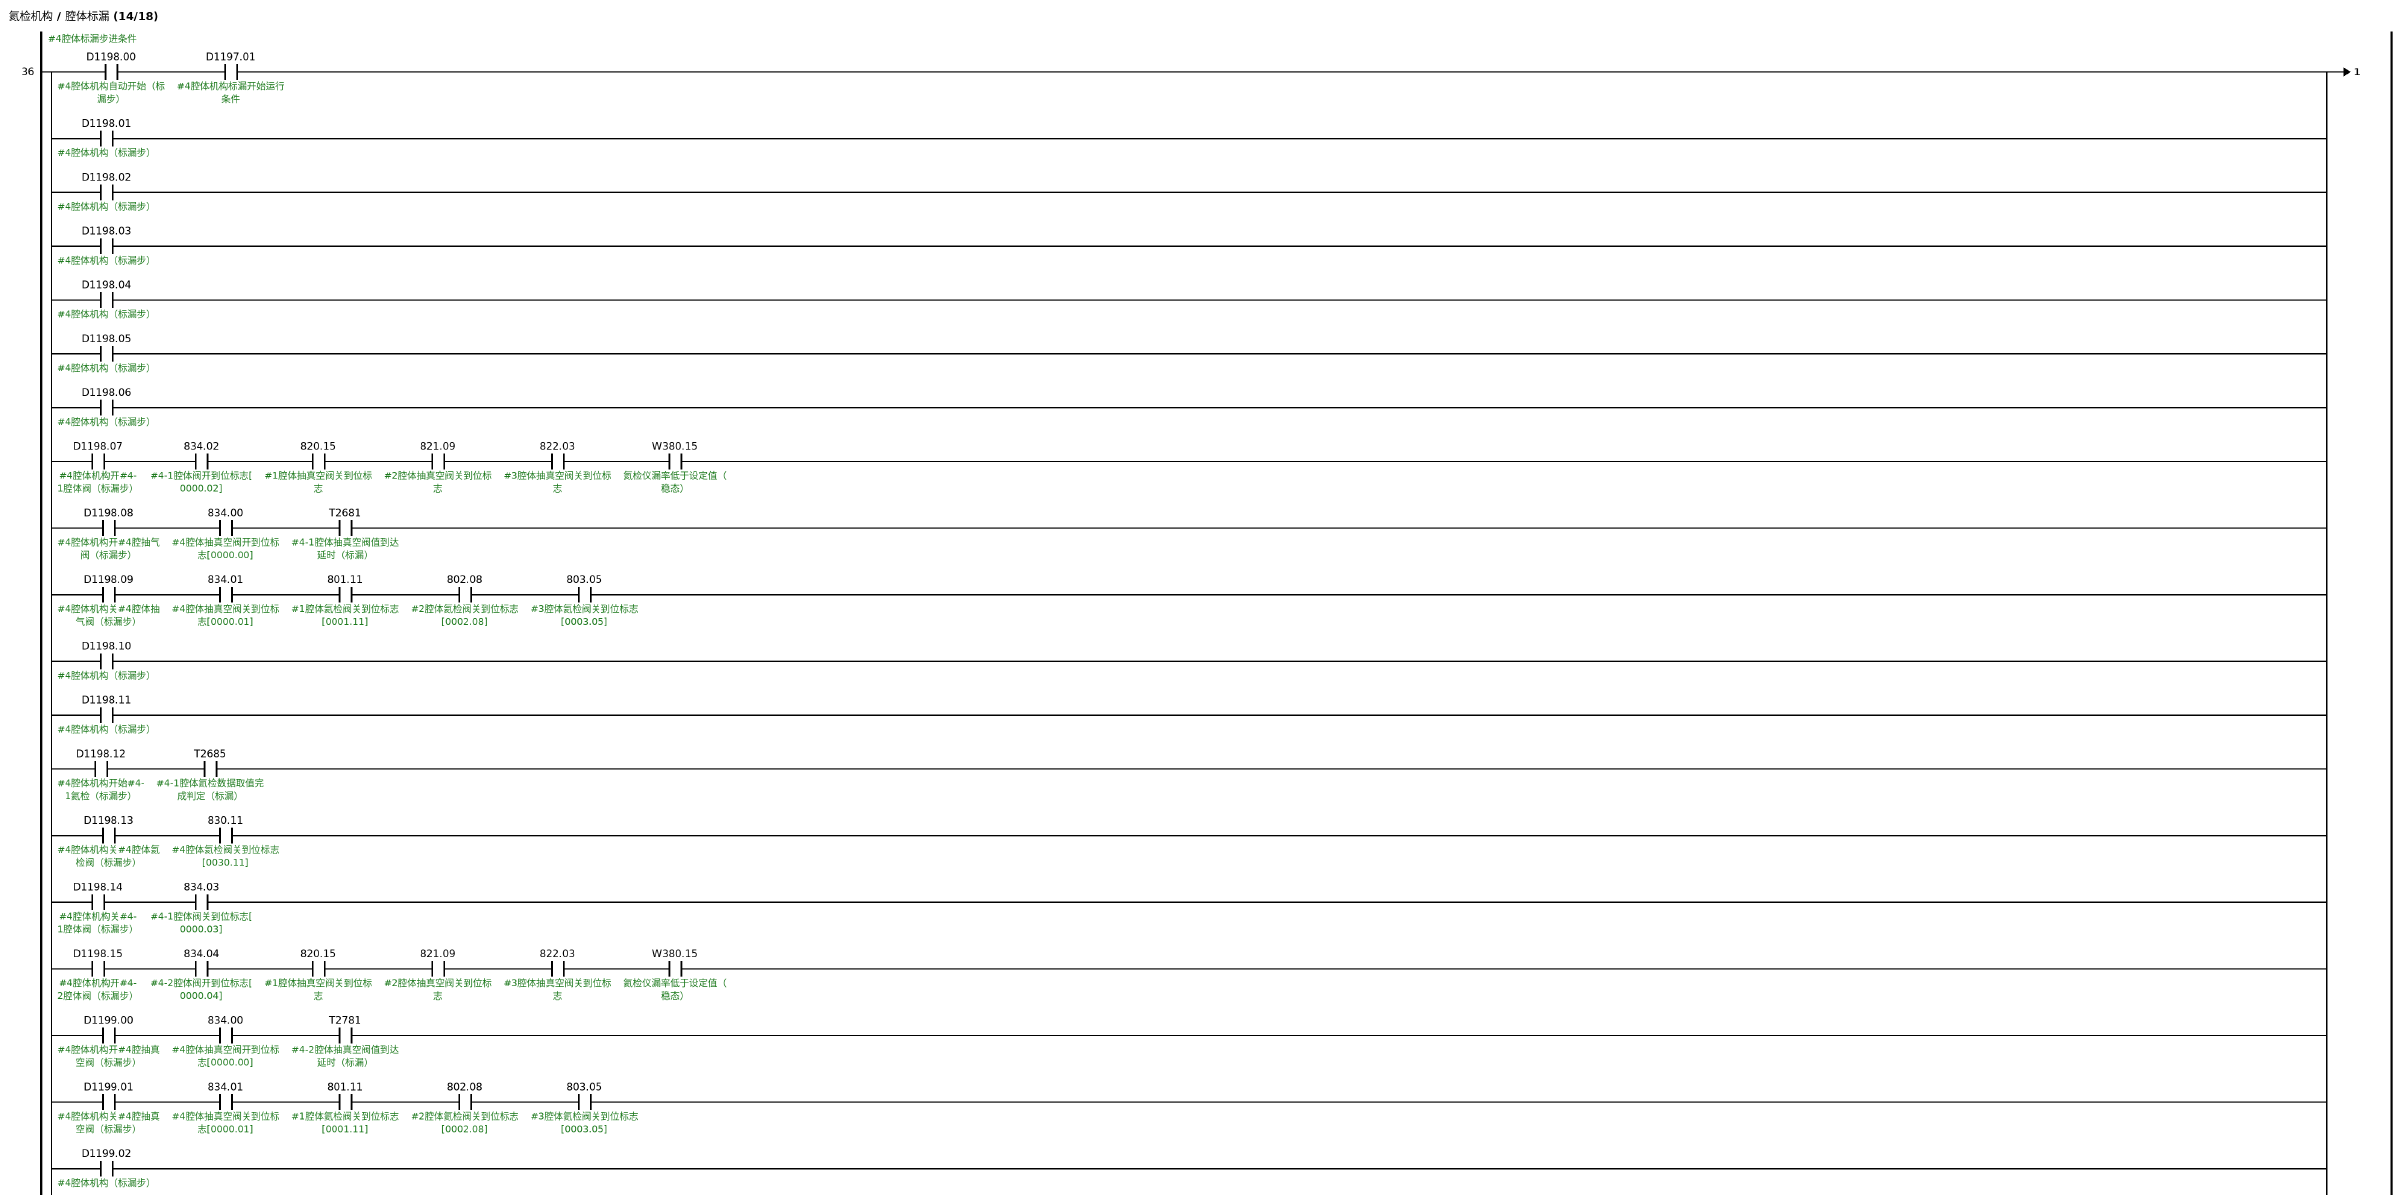

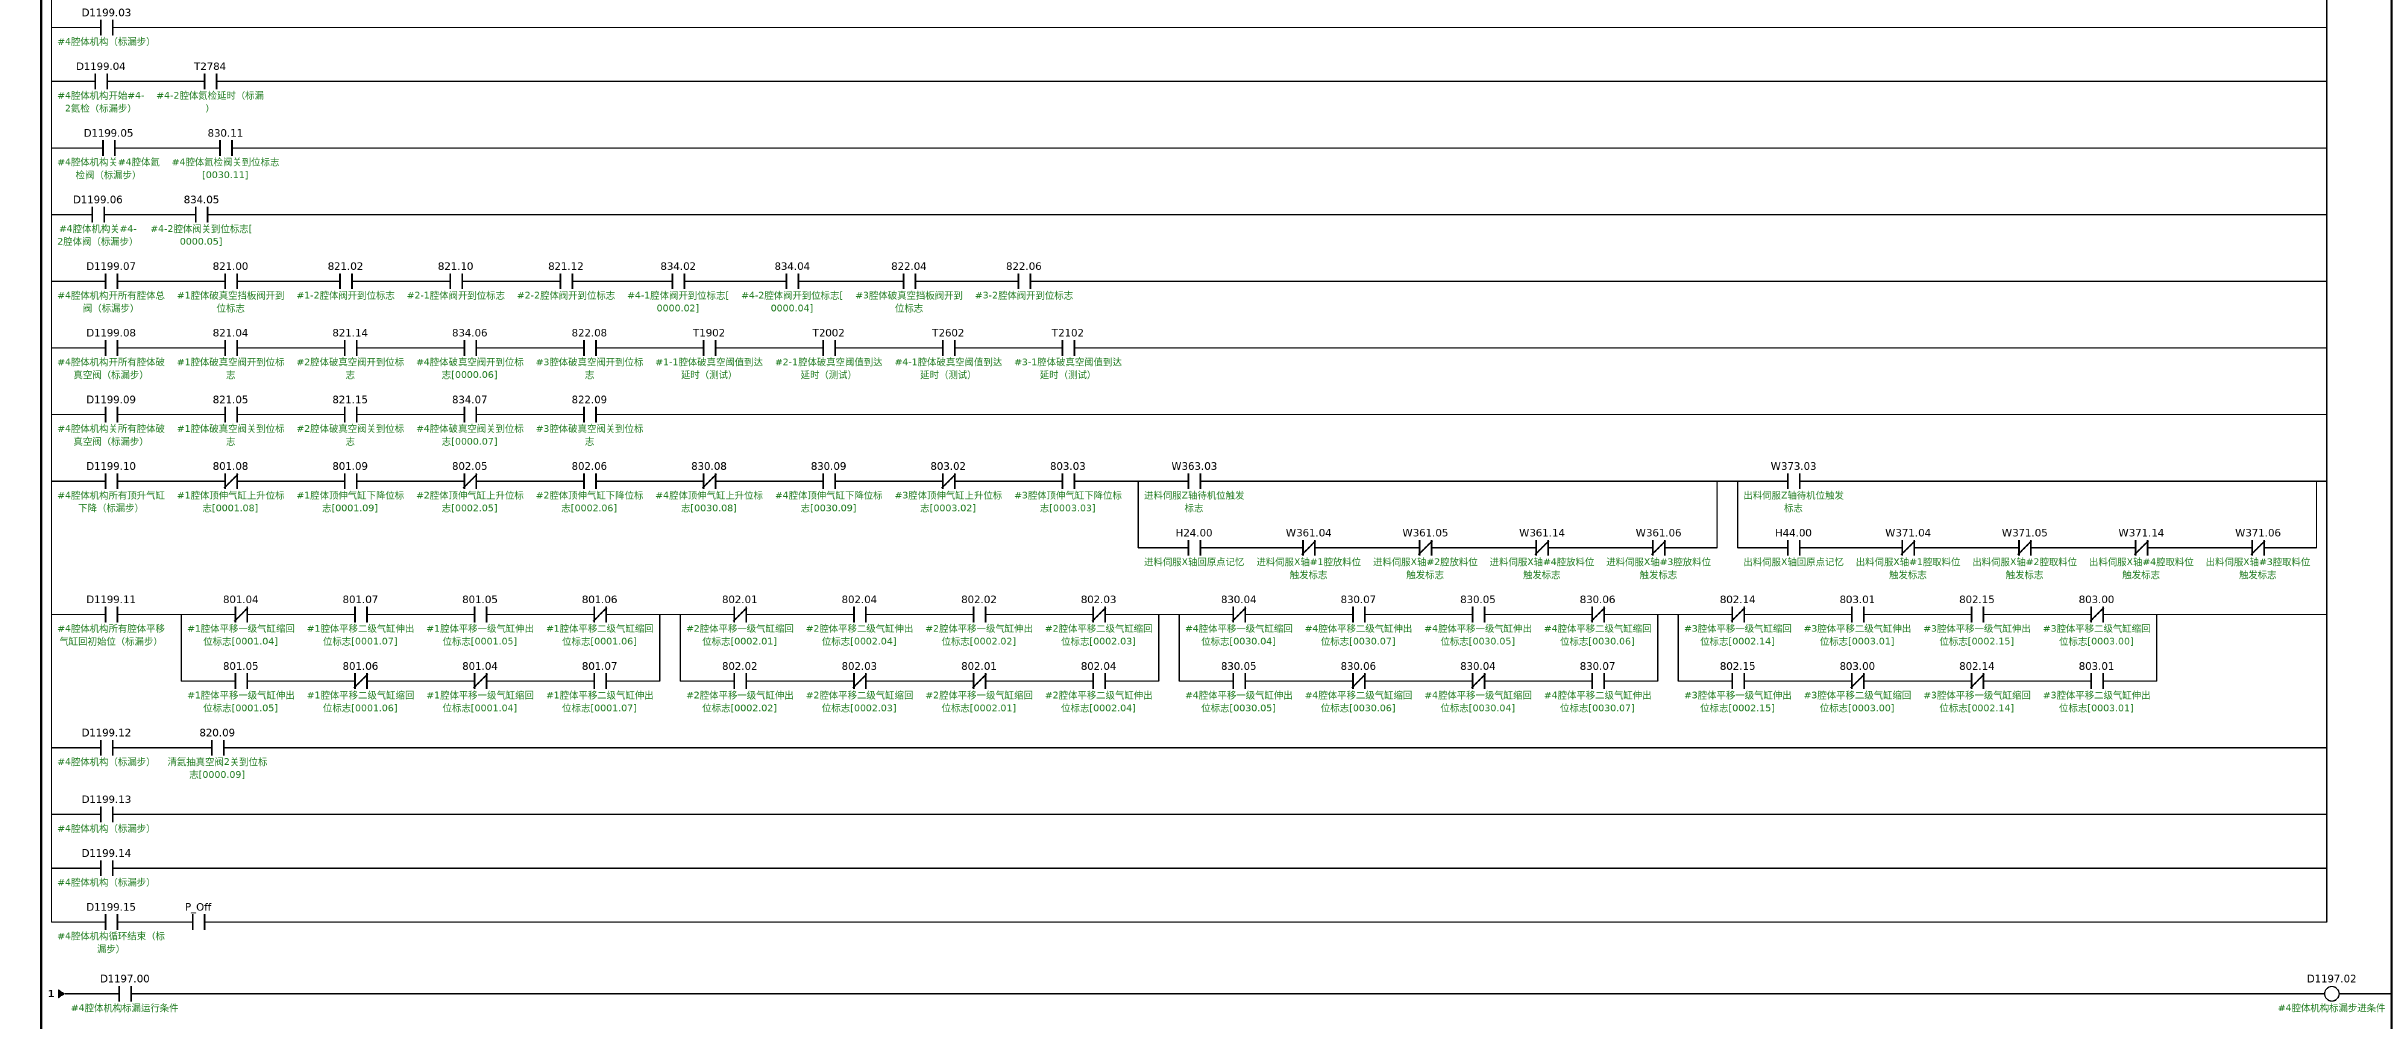
; rung 36: #4腔体标漏步进条件
LD D1198.00  ; #4腔体机构自动开始（标漏步）
AND D1197.01  ; #4腔体机构标漏开始运行条件
OR D1198.01  ; #4腔体机构（标漏步）
OR D1198.02  ; #4腔体机构（标漏步）
OR D1198.03  ; #4腔体机构（标漏步）
OR D1198.04  ; #4腔体机构（标漏步）
OR D1198.05  ; #4腔体机构（标漏步）
OR D1198.06  ; #4腔体机构（标漏步）
LD D1198.07  ; #4腔体机构开#4-1腔体阀（标漏步）
AND 834.02  ; #4-1腔体阀开到位标志[0000.02]
AND 820.15  ; #1腔体抽真空阀关到位标志
AND 821.09  ; #2腔体抽真空阀关到位标志
AND 822.03  ; #3腔体抽真空阀关到位标志
AND W380.15  ; 氦检仪漏率低于设定值（稳态）
ORLD
LD D1198.08  ; #4腔体机构开#4腔抽气阀（标漏步）
AND 834.00  ; #4腔体抽真空阀开到位标志[0000.00]
AND T2681  ; #4-1腔体抽真空阀值到达延时（标漏）
ORLD
LD D1198.09  ; #4腔体机构关#4腔体抽气阀（标漏步）
AND 834.01  ; #4腔体抽真空阀关到位标志[0000.01]
AND 801.11  ; #1腔体氦检阀关到位标志[0001.11]
AND 802.08  ; #2腔体氦检阀关到位标志[0002.08]
AND 803.05  ; #3腔体氦检阀关到位标志[0003.05]
ORLD
OR D1198.10  ; #4腔体机构（标漏步）
OR D1198.11  ; #4腔体机构（标漏步）
LD D1198.12  ; #4腔体机构开始#4-1氦检（标漏步）
AND T2685  ; #4-1腔体氦检数据取值完成判定（标漏）
ORLD
LD D1198.13  ; #4腔体机构关#4腔体氦检阀（标漏步）
AND 830.11  ; #4腔体氦检阀关到位标志[0030.11]
ORLD
LD D1198.14  ; #4腔体机构关#4-1腔体阀（标漏步）
AND 834.03  ; #4-1腔体阀关到位标志[0000.03]
ORLD
LD D1198.15  ; #4腔体机构开#4-2腔体阀（标漏步）
AND 834.04  ; #4-2腔体阀开到位标志[0000.04]
AND 820.15  ; #1腔体抽真空阀关到位标志
AND 821.09  ; #2腔体抽真空阀关到位标志
AND 822.03  ; #3腔体抽真空阀关到位标志
AND W380.15  ; 氦检仪漏率低于设定值（稳态）
ORLD
LD D1199.00  ; #4腔体机构开#4腔抽真空阀（标漏步）
AND 834.00  ; #4腔体抽真空阀开到位标志[0000.00]
AND T2781  ; #4-2腔体抽真空阀值到达延时（标漏）
ORLD
LD D1199.01  ; #4腔体机构关#4腔抽真空阀（标漏步）
AND 834.01  ; #4腔体抽真空阀关到位标志[0000.01]
AND 801.11  ; #1腔体氦检阀关到位标志[0001.11]
AND 802.08  ; #2腔体氦检阀关到位标志[0002.08]
AND 803.05  ; #3腔体氦检阀关到位标志[0003.05]
ORLD
OR D1199.02  ; #4腔体机构（标漏步）
OR D1199.03  ; #4腔体机构（标漏步）
LD D1199.04  ; #4腔体机构开始#4-2氦检（标漏步）
AND T2784  ; #4-2腔体氦检延时（标漏）
ORLD
LD D1199.05  ; #4腔体机构关#4腔体氦检阀（标漏步）
AND 830.11  ; #4腔体氦检阀关到位标志[0030.11]
ORLD
LD D1199.06  ; #4腔体机构关#4-2腔体阀（标漏步）
AND 834.05  ; #4-2腔体阀关到位标志[0000.05]
ORLD
LD D1199.07  ; #4腔体机构开所有腔体总阀（标漏步）
AND 821.00  ; #1腔体破真空挡板阀开到位标志
AND 821.02  ; #1-2腔体阀开到位标志
AND 821.10  ; #2-1腔体阀开到位标志
AND 821.12  ; #2-2腔体阀开到位标志
AND 834.02  ; #4-1腔体阀开到位标志[0000.02]
AND 834.04  ; #4-2腔体阀开到位标志[0000.04]
AND 822.04  ; #3腔体破真空挡板阀开到位标志
AND 822.06  ; #3-2腔体阀开到位标志
ORLD
LD D1199.08  ; #4腔体机构开所有腔体破真空阀（标漏步）
AND 821.04  ; #1腔体破真空阀开到位标志
AND 821.14  ; #2腔体破真空阀开到位标志
AND 834.06  ; #4腔体破真空阀开到位标志[0000.06]
AND 822.08  ; #3腔体破真空阀开到位标志
AND T1902  ; #1-1腔体破真空阈值到达延时（测试）
AND T2002  ; #2-1腔体破真空阈值到达延时（测试）
AND T2602  ; #4-1腔体破真空阈值到达延时（测试）
AND T2102  ; #3-1腔体破真空阈值到达延时（测试）
ORLD
LD D1199.09  ; #4腔体机构关所有腔体破真空阀（标漏步）
AND 821.05  ; #1腔体破真空阀关到位标志
AND 821.15  ; #2腔体破真空阀关到位标志
AND 834.07  ; #4腔体破真空阀关到位标志[0000.07]
AND 822.09  ; #3腔体破真空阀关到位标志
ORLD
LD D1199.10  ; #4腔体机构所有顶升气缸下降（标漏步）
ANDNOT 801.08  ; #1腔体顶伸气缸上升位标志[0001.08]
AND 801.09  ; #1腔体顶伸气缸下降位标志[0001.09]
ANDNOT 802.05  ; #2腔体顶伸气缸上升位标志[0002.05]
AND 802.06  ; #2腔体顶伸气缸下降位标志[0002.06]
ANDNOT 830.08  ; #4腔体顶伸气缸上升位标志[0030.08]
AND 830.09  ; #4腔体顶伸气缸下降位标志[0030.09]
ANDNOT 803.02  ; #3腔体顶伸气缸上升位标志[0003.02]
AND 803.03  ; #3腔体顶伸气缸下降位标志[0003.03]
LD W363.03  ; 进料伺服Z轴待机位触发标志
LD H24.00  ; 进料伺服X轴回原点记忆
ANDNOT W361.04  ; 进料伺服X轴#1腔放料位触发标志
ANDNOT W361.05  ; 进料伺服X轴#2腔放料位触发标志
ANDNOT W361.14  ; 进料伺服X轴#4腔放料位触发标志
ANDNOT W361.06  ; 进料伺服X轴#3腔放料位触发标志
ORLD
ANDLD
LD W373.03  ; 出料伺服Z轴待机位触发标志
LD H44.00  ; 出料伺服X轴回原点记忆
ANDNOT W371.04  ; 出料伺服X轴#1腔取料位触发标志
ANDNOT W371.05  ; 出料伺服X轴#2腔取料位触发标志
ANDNOT W371.14  ; 出料伺服X轴#4腔取料位触发标志
ANDNOT W371.06  ; 出料伺服X轴#3腔取料位触发标志
ORLD
ANDLD
ORLD
LD D1199.11  ; #4腔体机构所有腔体平移气缸回初始位（标漏步）
LDNOT 801.04  ; #1腔体平移一级气缸缩回位标志[0001.04]
AND 801.07  ; #1腔体平移二级气缸伸出位标志[0001.07]
AND 801.05  ; #1腔体平移一级气缸伸出位标志[0001.05]
ANDNOT 801.06  ; #1腔体平移二级气缸缩回位标志[0001.06]
LD 801.05  ; #1腔体平移一级气缸伸出位标志[0001.05]
ANDNOT 801.06  ; #1腔体平移二级气缸缩回位标志[0001.06]
ANDNOT 801.04  ; #1腔体平移一级气缸缩回位标志[0001.04]
AND 801.07  ; #1腔体平移二级气缸伸出位标志[0001.07]
ORLD
ANDLD
LDNOT 802.01  ; #2腔体平移一级气缸缩回位标志[0002.01]
AND 802.04  ; #2腔体平移二级气缸伸出位标志[0002.04]
AND 802.02  ; #2腔体平移一级气缸伸出位标志[0002.02]
ANDNOT 802.03  ; #2腔体平移二级气缸缩回位标志[0002.03]
LD 802.02  ; #2腔体平移一级气缸伸出位标志[0002.02]
ANDNOT 802.03  ; #2腔体平移二级气缸缩回位标志[0002.03]
ANDNOT 802.01  ; #2腔体平移一级气缸缩回位标志[0002.01]
AND 802.04  ; #2腔体平移二级气缸伸出位标志[0002.04]
ORLD
ANDLD
LDNOT 830.04  ; #4腔体平移一级气缸缩回位标志[0030.04]
AND 830.07  ; #4腔体平移二级气缸伸出位标志[0030.07]
AND 830.05  ; #4腔体平移一级气缸伸出位标志[0030.05]
ANDNOT 830.06  ; #4腔体平移二级气缸缩回位标志[0030.06]
LD 830.05  ; #4腔体平移一级气缸伸出位标志[0030.05]
ANDNOT 830.06  ; #4腔体平移二级气缸缩回位标志[0030.06]
ANDNOT 830.04  ; #4腔体平移一级气缸缩回位标志[0030.04]
AND 830.07  ; #4腔体平移二级气缸伸出位标志[0030.07]
ORLD
ANDLD
LDNOT 802.14  ; #3腔体平移一级气缸缩回位标志[0002.14]
AND 803.01  ; #3腔体平移二级气缸伸出位标志[0003.01]
AND 802.15  ; #3腔体平移一级气缸伸出位标志[0002.15]
ANDNOT 803.00  ; #3腔体平移二级气缸缩回位标志[0003.00]
LD 802.15  ; #3腔体平移一级气缸伸出位标志[0002.15]
ANDNOT 803.00  ; #3腔体平移二级气缸缩回位标志[0003.00]
ANDNOT 802.14  ; #3腔体平移一级气缸缩回位标志[0002.14]
AND 803.01  ; #3腔体平移二级气缸伸出位标志[0003.01]
ORLD
ANDLD
ORLD
LD D1199.12  ; #4腔体机构（标漏步）
AND 820.09  ; 清氦抽真空阀2关到位标志[0000.09]
ORLD
OR D1199.13  ; #4腔体机构（标漏步）
OR D1199.14  ; #4腔体机构（标漏步）
LD D1199.15  ; #4腔体机构循环结束（标漏步）
AND P_Off
ORLD
AND D1197.00  ; #4腔体机构标漏运行条件
OUT D1197.02  ; #4腔体机构标漏步进条件

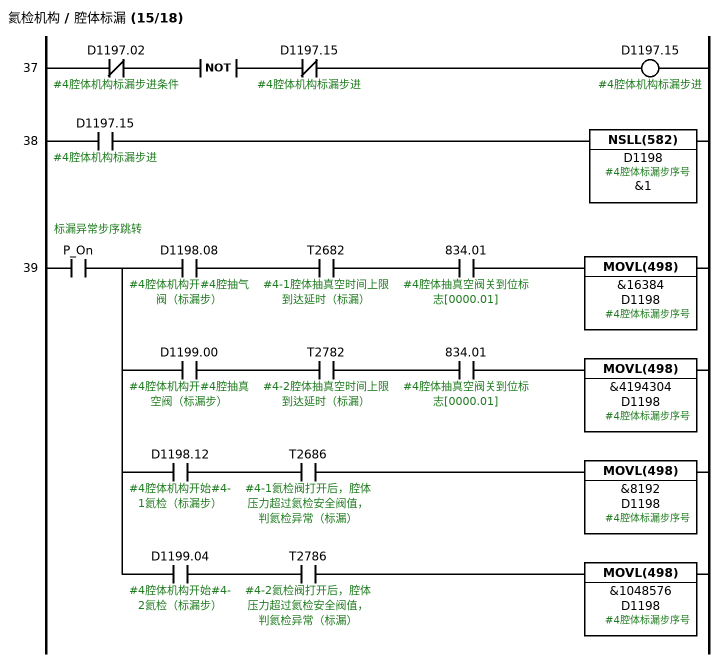
; rung 37
LDNOT D1197.02  ; #4腔体机构标漏步进条件
NOT(520)
ANDNOT D1197.15  ; #4腔体机构标漏步进
OUT D1197.15  ; #4腔体机构标漏步进
; rung 38
LD D1197.15  ; #4腔体机构标漏步进
NSLL(582) D1198 &1  ; #4腔体标漏步序号
; rung 39: 标漏异常步序跳转
LD P_On
OUT TR0
AND D1198.08  ; #4腔体机构开#4腔抽气阀（标漏步）
AND T2682  ; #4-1腔体抽真空时间上限到达延时（标漏）
AND 834.01  ; #4腔体抽真空阀关到位标志[0000.01]
MOVL(498) &16384 D1198  ; #4腔体标漏步序号
LD TR0
AND D1199.00  ; #4腔体机构开#4腔抽真空阀（标漏步）
AND T2782  ; #4-2腔体抽真空时间上限到达延时（标漏）
AND 834.01  ; #4腔体抽真空阀关到位标志[0000.01]
MOVL(498) &4194304 D1198  ; #4腔体标漏步序号
LD TR0
AND D1198.12  ; #4腔体机构开始#4-1氦检（标漏步）
AND T2686  ; #4-1氦检阀打开后，腔体压力超过氦检安全阀值，判氦检异常（标漏）
MOVL(498) &8192 D1198  ; #4腔体标漏步序号
LD TR0
AND D1199.04  ; #4腔体机构开始#4-2氦检（标漏步）
AND T2786  ; #4-2氦检阀打开后，腔体压力超过氦检安全阀值，判氦检异常（标漏）
MOVL(498) &1048576 D1198  ; #4腔体标漏步序号

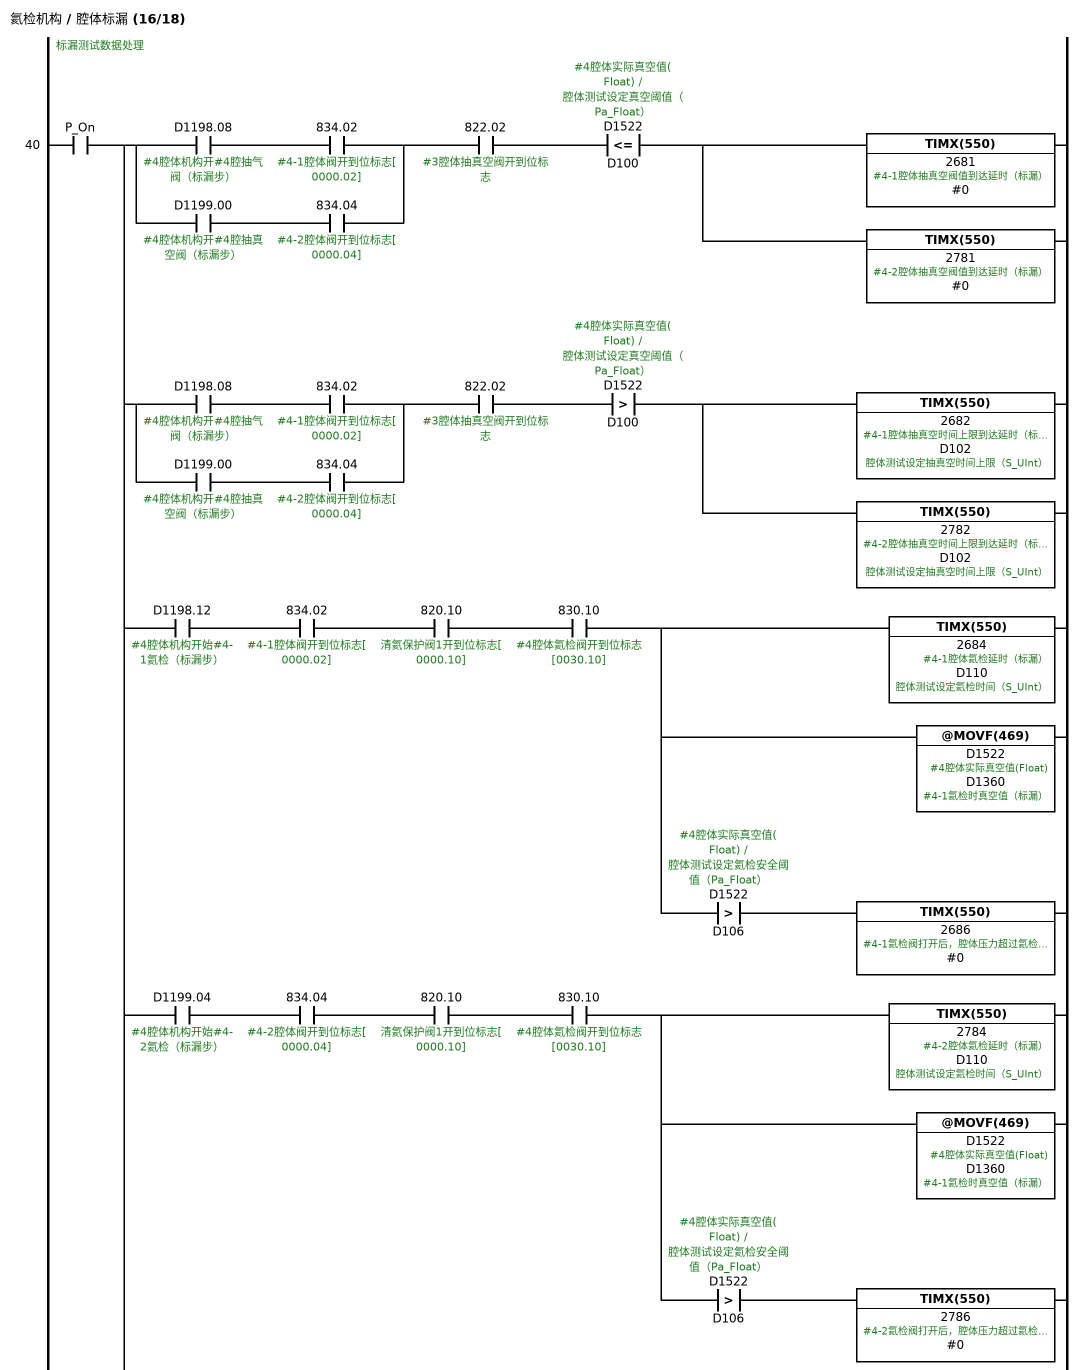

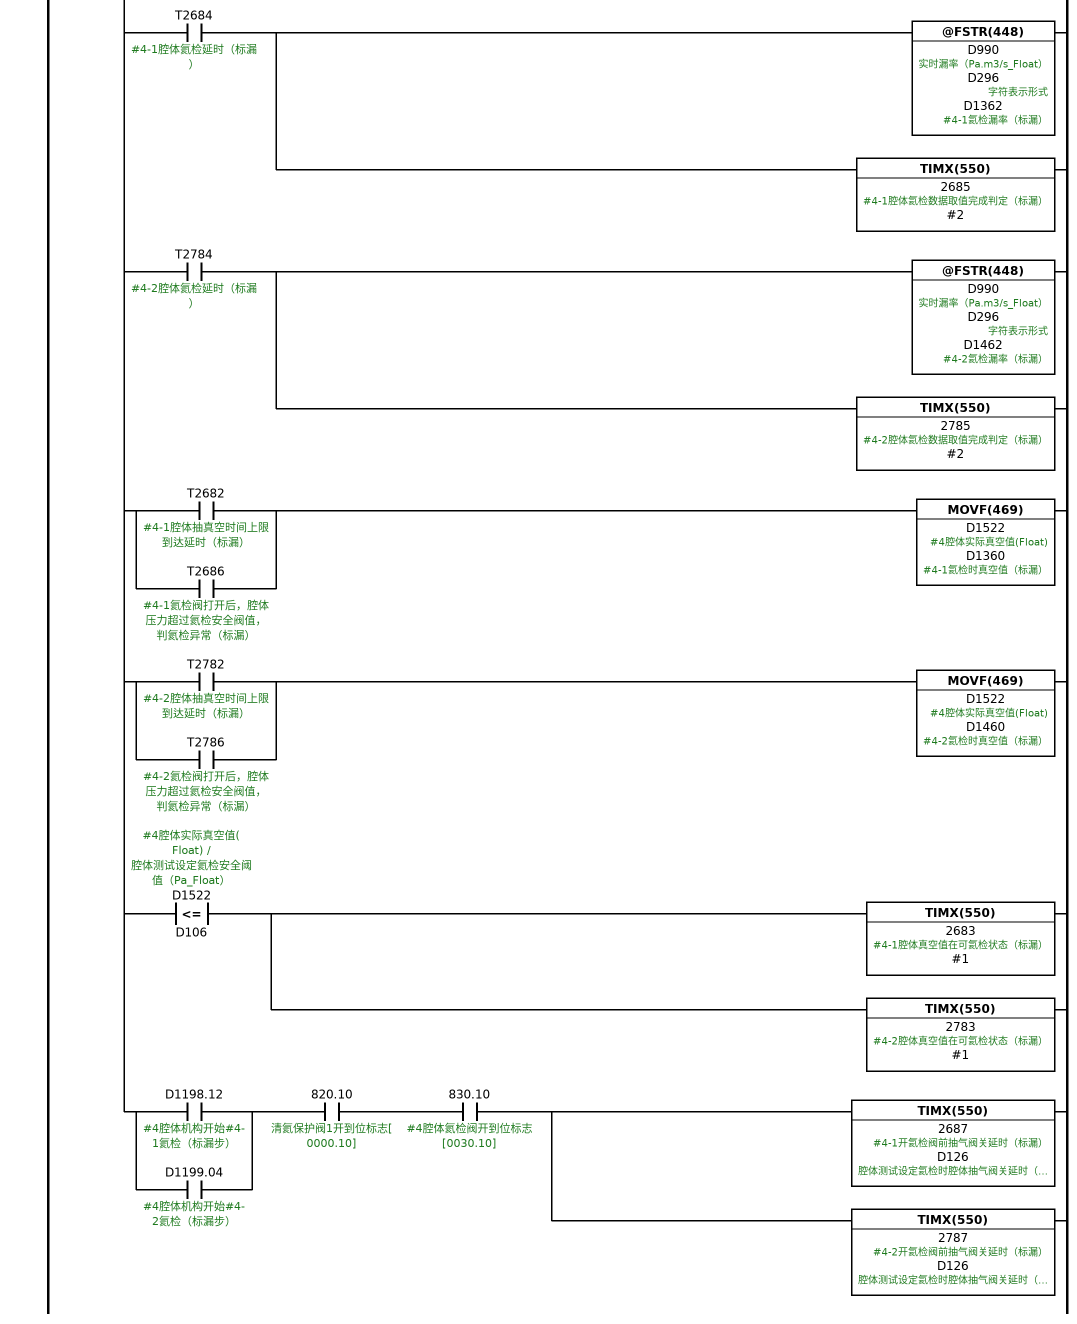
; rung 40: 标漏测试数据处理
LD P_On
OUT TR0
LD D1198.08  ; #4腔体机构开#4腔抽气阀（标漏步）
AND 834.02  ; #4-1腔体阀开到位标志[0000.02]
LD D1199.00  ; #4腔体机构开#4腔抽真空阀（标漏步）
AND 834.04  ; #4-2腔体阀开到位标志[0000.04]
ORLD
ANDLD
AND 822.02  ; #3腔体抽真空阀开到位标志
AND<=F(332) D1522 D100  ; #4腔体实际真空值(Float), 腔体测试设定真空阈值（Pa_Float）
TIMX(550) 2681 #0  ; #4-1腔体抽真空阀值到达延时（标漏）
TIMX(550) 2781 #0  ; #4-2腔体抽真空阀值到达延时（标漏）
LD TR0
LD D1198.08  ; #4腔体机构开#4腔抽气阀（标漏步）
AND 834.02  ; #4-1腔体阀开到位标志[0000.02]
LD D1199.00  ; #4腔体机构开#4腔抽真空阀（标漏步）
AND 834.04  ; #4-2腔体阀开到位标志[0000.04]
ORLD
ANDLD
AND 822.02  ; #3腔体抽真空阀开到位标志
AND>F(333) D1522 D100  ; #4腔体实际真空值(Float), 腔体测试设定真空阈值（Pa_Float）
TIMX(550) 2682 D102  ; 腔体测试设定抽真空时间上限（S_UInt）, #4-1腔体抽真空时间上限到达延时（标漏）
TIMX(550) 2782 D102  ; 腔体测试设定抽真空时间上限（S_UInt）, #4-2腔体抽真空时间上限到达延时（标漏）
LD TR0
AND D1198.12  ; #4腔体机构开始#4-1氦检（标漏步）
AND 834.02  ; #4-1腔体阀开到位标志[0000.02]
AND 820.10  ; 清氦保护阀1开到位标志[0000.10]
AND 830.10  ; #4腔体氦检阀开到位标志[0030.10]
TIMX(550) 2684 D110  ; 腔体测试设定氦检时间（S_UInt）, #4-1腔体氦检延时（标漏）
@MOVF(469) D1522 D1360  ; #4腔体实际真空值(Float), #4-1氦检时真空值（标漏）
AND>F(333) D1522 D106  ; #4腔体实际真空值(Float), 腔体测试设定氦检安全阈值（Pa_Float）
TIMX(550) 2686 #0  ; #4-1氦检阀打开后，腔体压力超过氦检安全阀值，判氦检异常（标漏）
LD TR0
AND D1199.04  ; #4腔体机构开始#4-2氦检（标漏步）
AND 834.04  ; #4-2腔体阀开到位标志[0000.04]
AND 820.10  ; 清氦保护阀1开到位标志[0000.10]
AND 830.10  ; #4腔体氦检阀开到位标志[0030.10]
TIMX(550) 2784 D110  ; 腔体测试设定氦检时间（S_UInt）, #4-2腔体氦检延时（标漏）
@MOVF(469) D1522 D1360  ; #4腔体实际真空值(Float), #4-1氦检时真空值（标漏）
AND>F(333) D1522 D106  ; #4腔体实际真空值(Float), 腔体测试设定氦检安全阈值（Pa_Float）
TIMX(550) 2786 #0  ; #4-2氦检阀打开后，腔体压力超过氦检安全阀值，判氦检异常（标漏）
LD TR0
AND T2684  ; #4-1腔体氦检延时（标漏）
@FSTR(448) D990 D296 D1362  ; 实时漏率（Pa.m3/s_Float）, 字符表示形式, #4-1氦检漏率（标漏）
TIMX(550) 2685 #2  ; #4-1腔体氦检数据取值完成判定（标漏）
LD TR0
AND T2784  ; #4-2腔体氦检延时（标漏）
@FSTR(448) D990 D296 D1462  ; 实时漏率（Pa.m3/s_Float）, 字符表示形式, #4-2氦检漏率（标漏）
TIMX(550) 2785 #2  ; #4-2腔体氦检数据取值完成判定（标漏）
LD TR0
LD T2682  ; #4-1腔体抽真空时间上限到达延时（标漏）
OR T2686  ; #4-1氦检阀打开后，腔体压力超过氦检安全阀值，判氦检异常（标漏）
ANDLD
MOVF(469) D1522 D1360  ; #4腔体实际真空值(Float), #4-1氦检时真空值（标漏）
LD TR0
LD T2782  ; #4-2腔体抽真空时间上限到达延时（标漏）
OR T2786  ; #4-2氦检阀打开后，腔体压力超过氦检安全阀值，判氦检异常（标漏）
ANDLD
MOVF(469) D1522 D1460  ; #4腔体实际真空值(Float), #4-2氦检时真空值（标漏）
LD TR0
AND<=F(332) D1522 D106  ; #4腔体实际真空值(Float), 腔体测试设定氦检安全阈值（Pa_Float）  // 未修改
TIMX(550) 2683 #1  ; #4-1腔体真空值在可氦检状态（标漏）
TIMX(550) 2783 #1  ; #4-2腔体真空值在可氦检状态（标漏）
LD TR0
LD D1198.12  ; #4腔体机构开始#4-1氦检（标漏步）
OR D1199.04  ; #4腔体机构开始#4-2氦检（标漏步）
ANDLD
AND 820.10  ; 清氦保护阀1开到位标志[0000.10]
AND 830.10  ; #4腔体氦检阀开到位标志[0030.10]
TIMX(550) 2687 D126  ; 腔体测试设定氦检时腔体抽气阀关延时（S_UInt）, #4-1开氦检阀前抽气阀关延时（标漏）
TIMX(550) 2787 D126  ; 腔体测试设定氦检时腔体抽气阀关延时（S_UInt）, #4-2开氦检阀前抽气阀关延时（标漏）

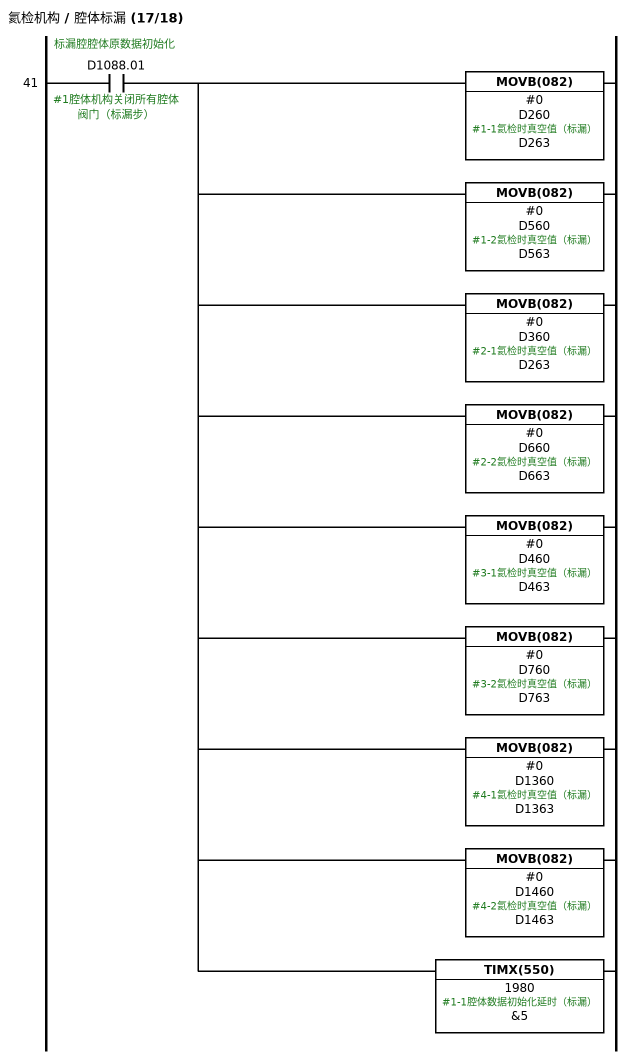
; rung 41: 标漏腔腔体原数据初始化
LD D1088.01  ; #1腔体机构关闭所有腔体阀门（标漏步）
MOVB(082) #0 D260 D263  ; #1-1氦检时真空值（标漏）
MOVB(082) #0 D560 D563  ; #1-2氦检时真空值（标漏）
MOVB(082) #0 D360 D263  ; #2-1氦检时真空值（标漏）
MOVB(082) #0 D660 D663  ; #2-2氦检时真空值（标漏）
MOVB(082) #0 D460 D463  ; #3-1氦检时真空值（标漏）
MOVB(082) #0 D760 D763  ; #3-2氦检时真空值（标漏）
MOVB(082) #0 D1360 D1363  ; #4-1氦检时真空值（标漏）
MOVB(082) #0 D1460 D1463  ; #4-2氦检时真空值（标漏）
TIMX(550) 1980 &5  ; #1-1腔体数据初始化延时（标漏）

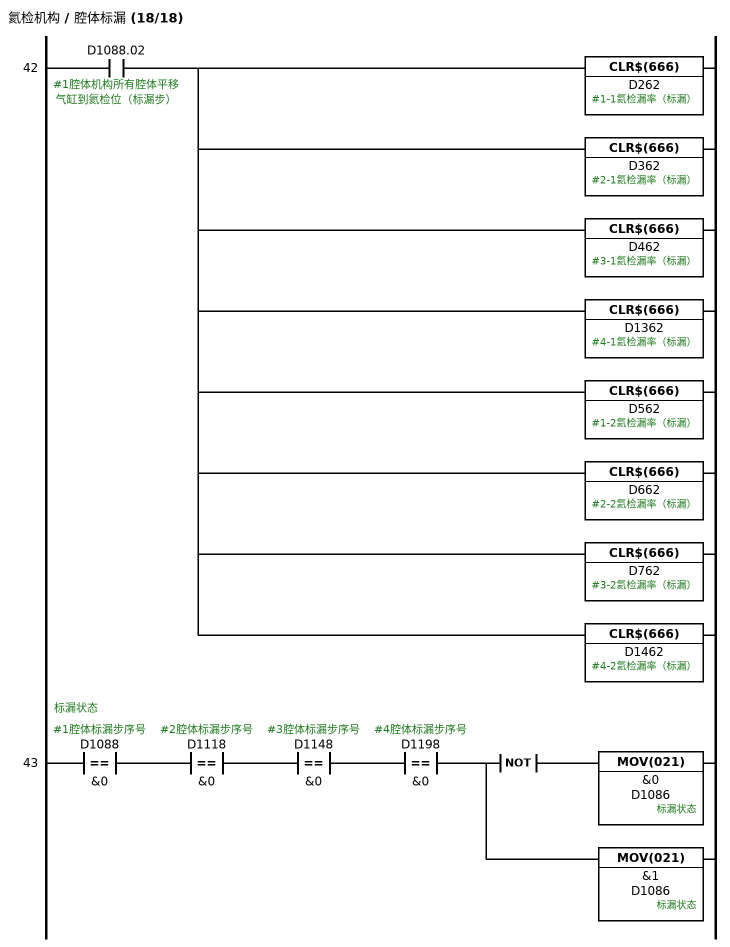
; rung 42
LD D1088.02  ; #1腔体机构所有腔体平移气缸到氦检位（标漏步）
CLR$(666) D262  ; #1-1氦检漏率（标漏）
CLR$(666) D362  ; #2-1氦检漏率（标漏）
CLR$(666) D462  ; #3-1氦检漏率（标漏）
CLR$(666) D1362  ; #4-1氦检漏率（标漏）
CLR$(666) D562  ; #1-2氦检漏率（标漏）
CLR$(666) D662  ; #2-2氦检漏率（标漏）
CLR$(666) D762  ; #3-2氦检漏率（标漏）
CLR$(666) D1462  ; #4-2氦检漏率（标漏）
; rung 43: 标漏状态
LD=L(301) D1088 &0  ; #1腔体标漏步序号
AND=L(301) D1118 &0  ; #2腔体标漏步序号
AND=L(301) D1148 &0  ; #3腔体标漏步序号
AND=L(301) D1198 &0  ; #4腔体标漏步序号
OUT TR0
NOT(520)
MOV(021) &0 D1086  ; 标漏状态
LD TR0
MOV(021) &1 D1086  ; 标漏状态

### Section 腔体自检

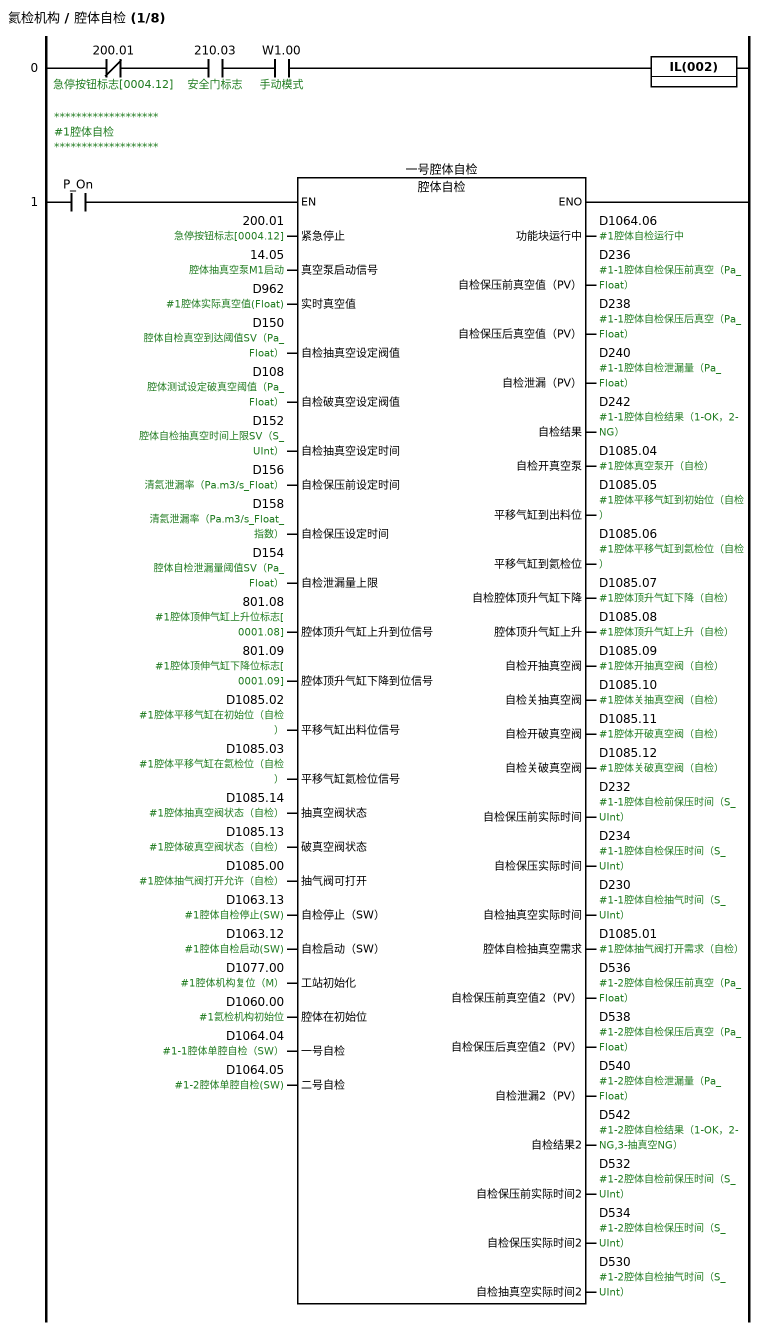
; rung 0
LDNOT 200.01  ; 急停按钮标志[0004.12]
AND 210.03  ; 安全门标志
AND W1.00  ; 手动模式
IL(002)
; rung 1: ******************* / #1腔体自检 / *******************
LD P_On
CALL 一号腔体自检 : 腔体自检 (紧急停止 := 200.01, 真空泵启动信号 := 14.05, 实时真空值 := D962, 自检抽真空设定阀值 := D150, 自检破真空设定阀值 := D108, 自检抽真空设定时间 := D152, 自检保压前设定时间 := D156, 自检保压设定时间 := D158, 自检泄漏量上限 := D154, 腔体顶升气缸上升到位信号 := 801.08, 腔体顶升气缸下降到位信号 := 801.09, 平移气缸出料位信号 := D1085.02, 平移气缸氦检位信号 := D1085.03, 抽真空阀状态 := D1085.14, 破真空阀状态 := D1085.13, 抽气阀可打开 := D1085.00, 自检停止（SW） := D1063.13, 自检启动（SW） := D1063.12, 工站初始化 := D1077.00, 腔体在初始位 := D1060.00, 一号自检 := D1064.04, 二号自检 := D1064.05, 功能块运行中 => D1064.06, 自检保压前真空值（PV） => D236, 自检保压后真空值（PV） => D238, 自检泄漏（PV） => D240, 自检结果 => D242, 自检开真空泵 => D1085.04, 平移气缸到出料位 => D1085.05, 平移气缸到氦检位 => D1085.06, 自检腔体顶升气缸下降 => D1085.07, 腔体顶升气缸上升 => D1085.08, 自检开抽真空阀 => D1085.09, 自检关抽真空阀 => D1085.10, 自检开破真空阀 => D1085.11, 自检关破真空阀 => D1085.12, 自检保压前实际时间 => D232, 自检保压实际时间 => D234, 自检抽真空实际时间 => D230, 腔体自检抽真空需求 => D1085.01, 自检保压前真空值2（PV） => D536, 自检保压后真空值2（PV） => D538, 自检泄漏2（PV） => D540, 自检结果2 => D542, 自检保压前实际时间2 => D532, 自检保压实际时间2 => D534, 自检抽真空实际时间2 => D530)  ; 急停按钮标志[0004.12], 腔体抽真空泵M1启动, #1腔体实际真空值(Float), 腔体自检真空到达阈值SV（Pa_Float）, 腔体测试设定破真空阈值（Pa_Float）, 腔体自检抽真空时间上限SV（S_UInt）, 清氦泄漏率（Pa.m3/s_Float）, 清氦泄漏率（Pa.m3/s_Float_指数）, 腔体自检泄漏量阈值SV（Pa_Float）, #1腔体顶伸气缸上升位标志[0001.08], #1腔体顶伸气缸下降位标志[0001.09], #1腔体平移气缸在初始位（自检）, #1腔体平移气缸在氦检位（自检）, #1腔体抽真空阀状态（自检）, #1腔体破真空阀状态（自检）, #1腔体抽气阀打开允许（自检）, #1腔体自检停止(SW), #1腔体自检启动(SW), #1腔体机构复位（M）, #1氦检机构初始位, #1-1腔体单腔自检（SW）, #1-2腔体单腔自检(SW), #1腔体自检运行中, #1-1腔体自检保压前真空（Pa_Float）, #1-1腔体自检保压后真空（Pa_Float）, #1-1腔体自检泄漏量（Pa_Float）, #1-1腔体自检结果（1-OK，2-NG）, #1腔体真空泵开（自检）, #1腔体平移气缸到初始位（自检）, #1腔体平移气缸到氦检位（自检）, #1腔体顶升气缸下降（自检）, #1腔体顶升气缸上升（自检）, #1腔体开抽真空阀（自检）, #1腔体关抽真空阀（自检）, #1腔体开破真空阀（自检）, #1腔体关破真空阀（自检）, #1-1腔体自检前保压时间（S_UInt）, #1-1腔体自检保压时间（S_UInt）, #1-1腔体自检抽气时间（S_UInt）, #1腔体抽气阀打开需求（自检）, #1-2腔体自检保压前真空（Pa_Float）, #1-2腔体自检保压后真空（Pa_Float）, #1-2腔体自检泄漏量（Pa_Float）, #1-2腔体自检结果（1-OK，2-NG,3-抽真空NG）, #1-2腔体自检前保压时间（S_UInt）, #1-2腔体自检保压时间（S_UInt）, #1-2腔体自检抽气时间（S_UInt）

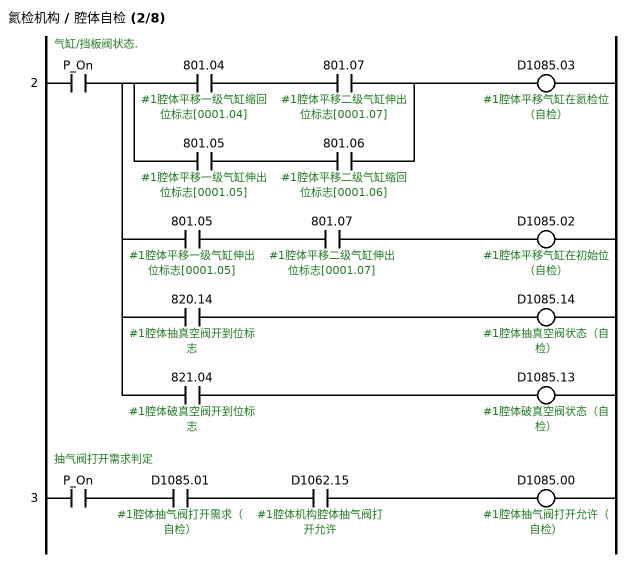
; rung 2: 气缸/挡板阀状态.
LD P_On
OUT TR0
LD 801.04  ; #1腔体平移一级气缸缩回位标志[0001.04]
AND 801.07  ; #1腔体平移二级气缸伸出位标志[0001.07]
LD 801.05  ; #1腔体平移一级气缸伸出位标志[0001.05]
AND 801.06  ; #1腔体平移二级气缸缩回位标志[0001.06]
ORLD
ANDLD
OUT D1085.03  ; #1腔体平移气缸在氦检位（自检）
LD TR0
AND 801.05  ; #1腔体平移一级气缸伸出位标志[0001.05]
AND 801.07  ; #1腔体平移二级气缸伸出位标志[0001.07]
OUT D1085.02  ; #1腔体平移气缸在初始位（自检）
LD TR0
AND 820.14  ; #1腔体抽真空阀开到位标志
OUT D1085.14  ; #1腔体抽真空阀状态（自检）
LD TR0
AND 821.04  ; #1腔体破真空阀开到位标志
OUT D1085.13  ; #1腔体破真空阀状态（自检）
; rung 3: 抽气阀打开需求判定
LD P_On
AND D1085.01  ; #1腔体抽气阀打开需求（自检）
AND D1062.15  ; #1腔体机构腔体抽气阀打开允许
OUT D1085.00  ; #1腔体抽气阀打开允许（自检）

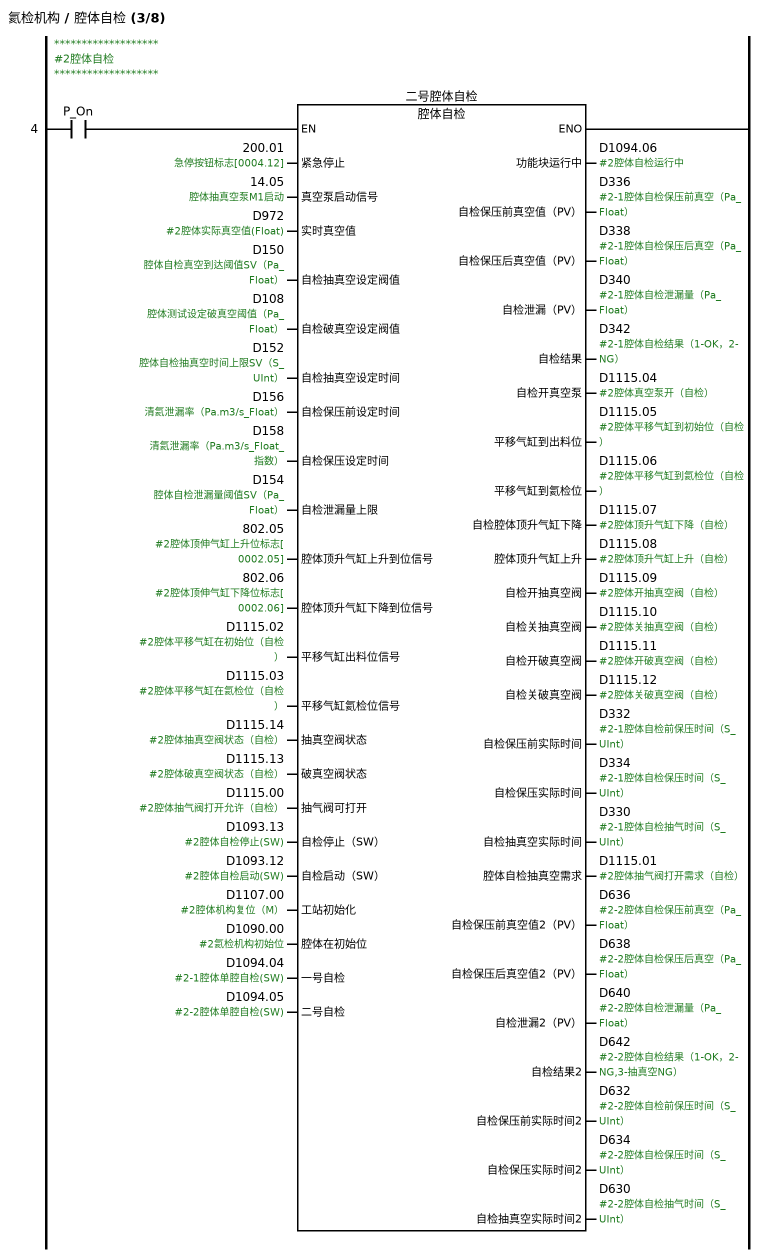
; rung 4: ******************* / #2腔体自检 / *******************
LD P_On
CALL 二号腔体自检 : 腔体自检 (紧急停止 := 200.01, 真空泵启动信号 := 14.05, 实时真空值 := D972, 自检抽真空设定阀值 := D150, 自检破真空设定阀值 := D108, 自检抽真空设定时间 := D152, 自检保压前设定时间 := D156, 自检保压设定时间 := D158, 自检泄漏量上限 := D154, 腔体顶升气缸上升到位信号 := 802.05, 腔体顶升气缸下降到位信号 := 802.06, 平移气缸出料位信号 := D1115.02, 平移气缸氦检位信号 := D1115.03, 抽真空阀状态 := D1115.14, 破真空阀状态 := D1115.13, 抽气阀可打开 := D1115.00, 自检停止（SW） := D1093.13, 自检启动（SW） := D1093.12, 工站初始化 := D1107.00, 腔体在初始位 := D1090.00, 一号自检 := D1094.04, 二号自检 := D1094.05, 功能块运行中 => D1094.06, 自检保压前真空值（PV） => D336, 自检保压后真空值（PV） => D338, 自检泄漏（PV） => D340, 自检结果 => D342, 自检开真空泵 => D1115.04, 平移气缸到出料位 => D1115.05, 平移气缸到氦检位 => D1115.06, 自检腔体顶升气缸下降 => D1115.07, 腔体顶升气缸上升 => D1115.08, 自检开抽真空阀 => D1115.09, 自检关抽真空阀 => D1115.10, 自检开破真空阀 => D1115.11, 自检关破真空阀 => D1115.12, 自检保压前实际时间 => D332, 自检保压实际时间 => D334, 自检抽真空实际时间 => D330, 腔体自检抽真空需求 => D1115.01, 自检保压前真空值2（PV） => D636, 自检保压后真空值2（PV） => D638, 自检泄漏2（PV） => D640, 自检结果2 => D642, 自检保压前实际时间2 => D632, 自检保压实际时间2 => D634, 自检抽真空实际时间2 => D630)  ; 急停按钮标志[0004.12], 腔体抽真空泵M1启动, #2腔体实际真空值(Float), 腔体自检真空到达阈值SV（Pa_Float）, 腔体测试设定破真空阈值（Pa_Float）, 腔体自检抽真空时间上限SV（S_UInt）, 清氦泄漏率（Pa.m3/s_Float）, 清氦泄漏率（Pa.m3/s_Float_指数）, 腔体自检泄漏量阈值SV（Pa_Float）, #2腔体顶伸气缸上升位标志[0002.05], #2腔体顶伸气缸下降位标志[0002.06], #2腔体平移气缸在初始位（自检）, #2腔体平移气缸在氦检位（自检）, #2腔体抽真空阀状态（自检）, #2腔体破真空阀状态（自检）, #2腔体抽气阀打开允许（自检）, #2腔体自检停止(SW), #2腔体自检启动(SW), #2腔体机构复位（M）, #2氦检机构初始位, #2-1腔体单腔自检(SW), #2-2腔体单腔自检(SW), #2腔体自检运行中, #2-1腔体自检保压前真空（Pa_Float）, #2-1腔体自检保压后真空（Pa_Float）, #2-1腔体自检泄漏量（Pa_Float）, #2-1腔体自检结果（1-OK，2-NG）, #2腔体真空泵开（自检）, #2腔体平移气缸到初始位（自检）, #2腔体平移气缸到氦检位（自检）, #2腔体顶升气缸下降（自检）, #2腔体顶升气缸上升（自检）, #2腔体开抽真空阀（自检）, #2腔体关抽真空阀（自检）, #2腔体开破真空阀（自检）, #2腔体关破真空阀（自检）, #2-1腔体自检前保压时间（S_UInt）, #2-1腔体自检保压时间（S_UInt）, #2-1腔体自检抽气时间（S_UInt）, #2腔体抽气阀打开需求（自检）, #2-2腔体自检保压前真空（Pa_Float）, #2-2腔体自检保压后真空（Pa_Float）, #2-2腔体自检泄漏量（Pa_Float）, #2-2腔体自检结果（1-OK，2-NG,3-抽真空NG）, #2-2腔体自检前保压时间（S_UInt）, #2-2腔体自检保压时间（S_UInt）, #2-2腔体自检抽气时间（S_UInt）

